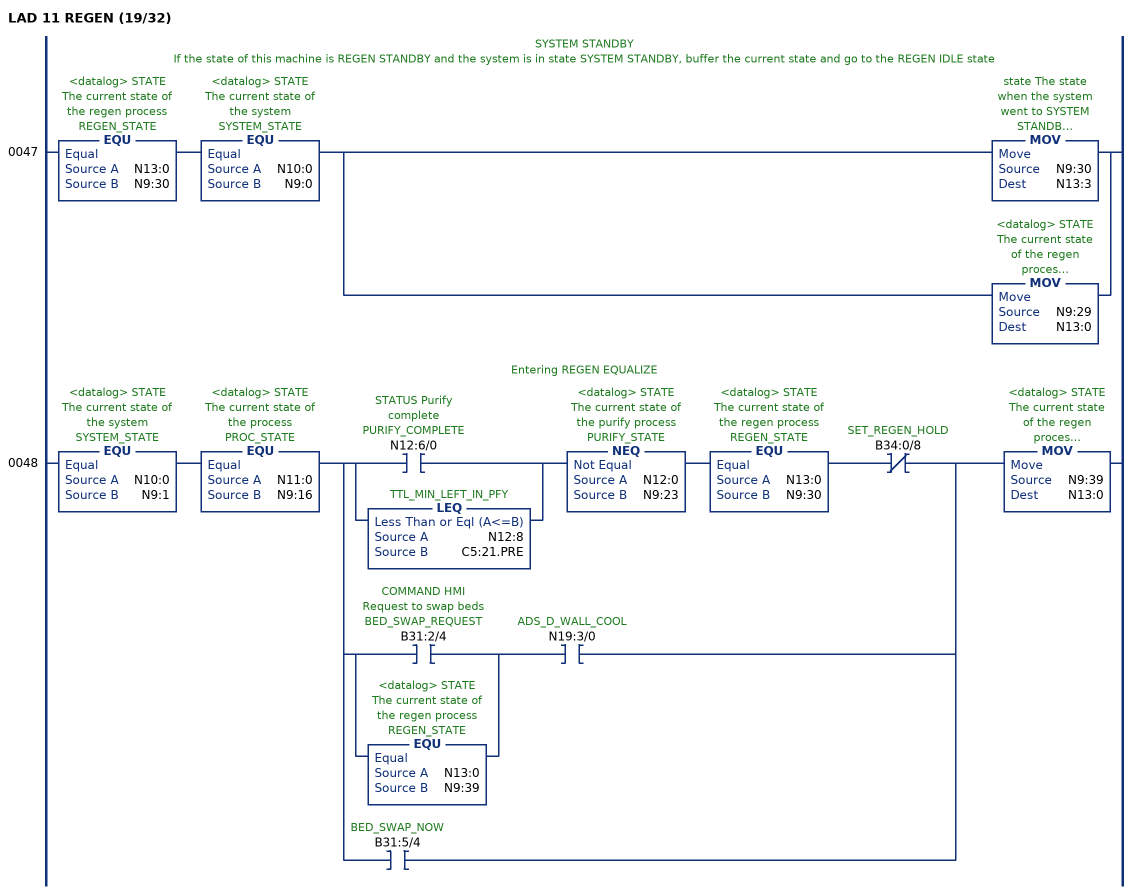
% Rung: 47 %
% SYSTEM STANDBY
% If the state of this machine is REGEN STANDBY and the system is in state SYSTEM STANDBY, buffer the current state and go to the REGEN IDLE state %
SOR EQU N13:0 N9:30 EQU N10:0 N9:0 BST MOV N9:30 N13:3 NXB MOV N9:29 N13:0 BND EOR
%   N13:0  REGEN_STATE  "<datalog> STATE The current state of the regen process" %
%   N9:30  REGEN_STANDBY  "STATE Regen Standby" %
%   N10:0  SYSTEM_STATE  "<datalog> STATE The current state of the system" %
%   N9:0  SYSTEM_STANDBY  "STATE System Standby" %
%   N13:3  REGEN_STANDBY_BUFFER  "state The state when the system went to SYSTEM STANDBY" %
%   N9:29  REGEN_IDLE  "STATE Regen Idle" %
% Rung: 48 %
% Entering REGEN EQUALIZE %
SOR EQU N10:0 N9:1 EQU N11:0 N9:16 BST BST XIC N12:6/0 NXB LEQ N12:8 C5:21.PRE BND NEQ N12:0 N9:23 EQU N13:0 N9:30 XIO B34:0/8 NXB BST XIC B31:2/4 NXB EQU N13:0 N9:39 BND XIC N19:3/0 NXB XIC B31:5/4 BND MOV N9:39 N13:0 EOR
%   N10:0  SYSTEM_STATE  "<datalog> STATE The current state of the system" %
%   N9:1  SYSTEM_PROCESS  "STATE System Process" %
%   N11:0  PROC_STATE  "<datalog> STATE The current state of the process" %
%   N9:16  PROC_REGEN_D  "STATE Process Regen D" %
%   N12:6/0  PURIFY_COMPLETE  "STATUS Purify complete" %
%   N12:8  TTL_MIN_LEFT_IN_PFY %
%   C5:21.PRE  "COUNTER Regen Equalize Time" %
%   N12:0  PURIFY_STATE  "<datalog> STATE The current state of the purify process" %
%   N9:23  PURIFY_MANUAL_HOLD  "STATE Purify Manual Hold" %
%   N13:0  REGEN_STATE  "<datalog> STATE The current state of the regen process" %
%   N9:30  REGEN_STANDBY  "STATE Regen Standby" %
%   B34:0/8  SET_REGEN_HOLD %
%   B31:2/4  BED_SWAP_REQUEST  "COMMAND HMI Request to swap beds" %
%   N9:39  REGEN_EQUALIZE  "STATE Regen Equalize" %
%   N19:3/0  ADS_D_WALL_COOL %
%   B31:5/4  BED_SWAP_NOW %

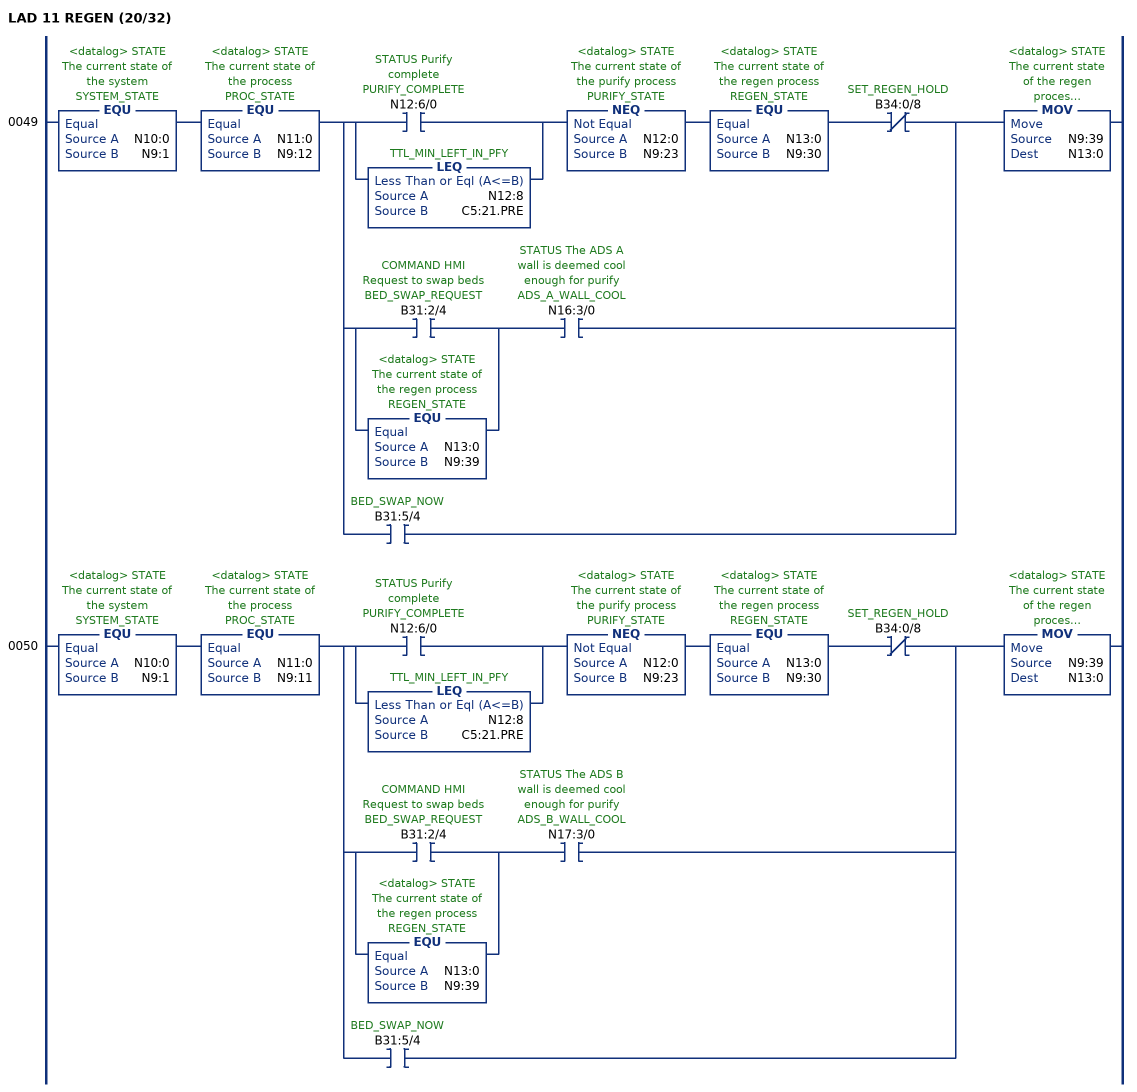
% Rung: 49 %
SOR EQU N10:0 N9:1 EQU N11:0 N9:12 BST BST XIC N12:6/0 NXB LEQ N12:8 C5:21.PRE BND NEQ N12:0 N9:23 EQU N13:0 N9:30 XIO B34:0/8 NXB BST XIC B31:2/4 NXB EQU N13:0 N9:39 BND XIC N16:3/0 NXB XIC B31:5/4 BND MOV N9:39 N13:0 EOR
%   N10:0  SYSTEM_STATE  "<datalog> STATE The current state of the system" %
%   N9:1  SYSTEM_PROCESS  "STATE System Process" %
%   N11:0  PROC_STATE  "<datalog> STATE The current state of the process" %
%   N9:12  PROC_REGEN_A  "STATE Process Regen A" %
%   N12:6/0  PURIFY_COMPLETE  "STATUS Purify complete" %
%   N12:8  TTL_MIN_LEFT_IN_PFY %
%   C5:21.PRE  "COUNTER Regen Equalize Time" %
%   N12:0  PURIFY_STATE  "<datalog> STATE The current state of the purify process" %
%   N9:23  PURIFY_MANUAL_HOLD  "STATE Purify Manual Hold" %
%   N13:0  REGEN_STATE  "<datalog> STATE The current state of the regen process" %
%   N9:30  REGEN_STANDBY  "STATE Regen Standby" %
%   B34:0/8  SET_REGEN_HOLD %
%   B31:2/4  BED_SWAP_REQUEST  "COMMAND HMI Request to swap beds" %
%   N9:39  REGEN_EQUALIZE  "STATE Regen Equalize" %
%   N16:3/0  ADS_A_WALL_COOL  "STATUS The ADS A wall is deemed cool enough for purify" %
%   B31:5/4  BED_SWAP_NOW %
% Rung: 50 %
SOR EQU N10:0 N9:1 EQU N11:0 N9:11 BST BST XIC N12:6/0 NXB LEQ N12:8 C5:21.PRE BND NEQ N12:0 N9:23 EQU N13:0 N9:30 XIO B34:0/8 NXB BST XIC B31:2/4 NXB EQU N13:0 N9:39 BND XIC N17:3/0 NXB XIC B31:5/4 BND MOV N9:39 N13:0 EOR
%   N10:0  SYSTEM_STATE  "<datalog> STATE The current state of the system" %
%   N9:1  SYSTEM_PROCESS  "STATE System Process" %
%   N11:0  PROC_STATE  "<datalog> STATE The current state of the process" %
%   N9:11  PROC_REGEN_B  "STATE Process Regen B" %
%   N12:6/0  PURIFY_COMPLETE  "STATUS Purify complete" %
%   N12:8  TTL_MIN_LEFT_IN_PFY %
%   C5:21.PRE  "COUNTER Regen Equalize Time" %
%   N12:0  PURIFY_STATE  "<datalog> STATE The current state of the purify process" %
%   N9:23  PURIFY_MANUAL_HOLD  "STATE Purify Manual Hold" %
%   N13:0  REGEN_STATE  "<datalog> STATE The current state of the regen process" %
%   N9:30  REGEN_STANDBY  "STATE Regen Standby" %
%   B34:0/8  SET_REGEN_HOLD %
%   B31:2/4  BED_SWAP_REQUEST  "COMMAND HMI Request to swap beds" %
%   N9:39  REGEN_EQUALIZE  "STATE Regen Equalize" %
%   N17:3/0  ADS_B_WALL_COOL  "STATUS The ADS B wall is deemed cool enough for purify" %
%   B31:5/4  BED_SWAP_NOW %

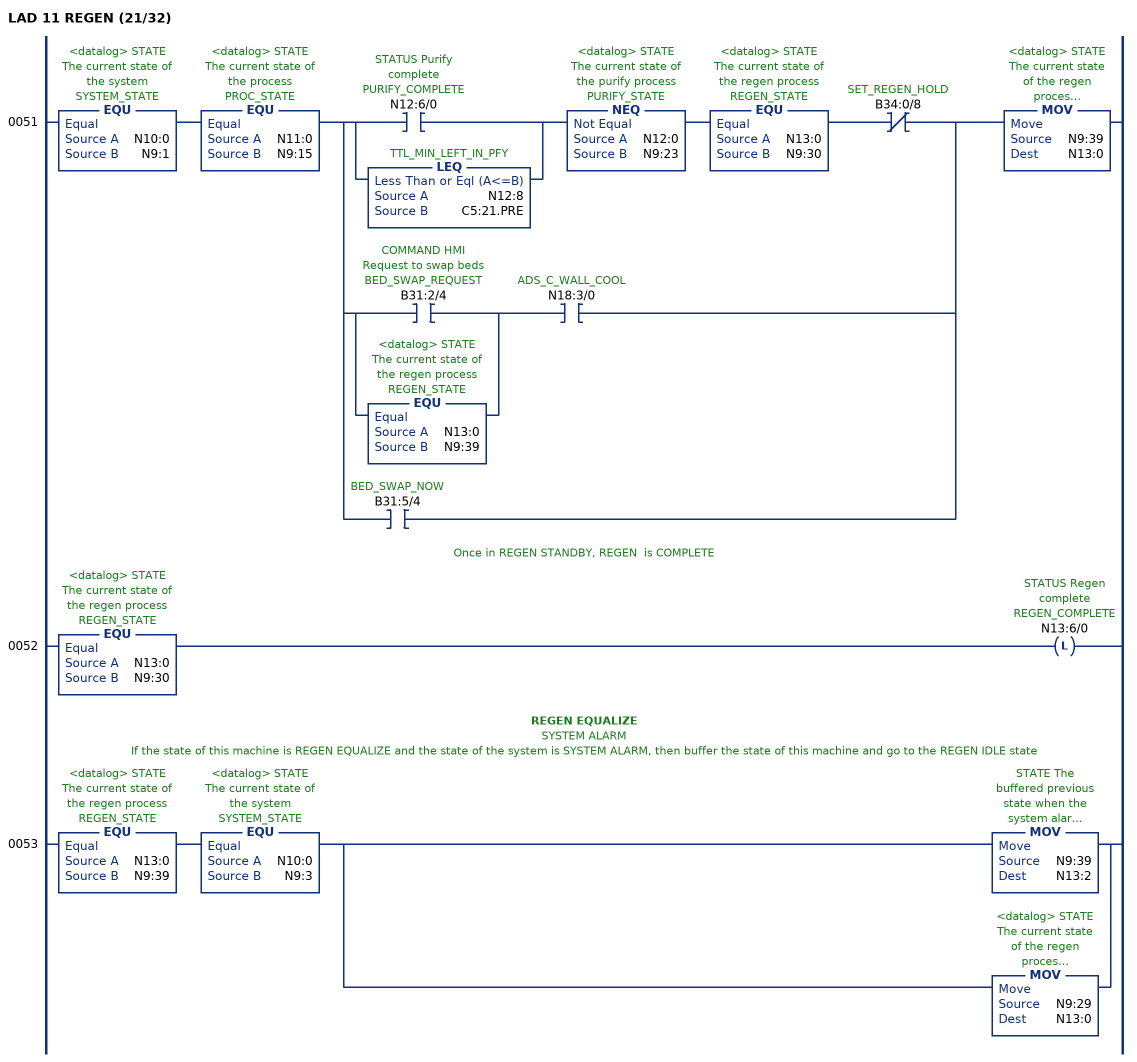
% Rung: 51 %
SOR EQU N10:0 N9:1 EQU N11:0 N9:15 BST BST XIC N12:6/0 NXB LEQ N12:8 C5:21.PRE BND NEQ N12:0 N9:23 EQU N13:0 N9:30 XIO B34:0/8 NXB BST XIC B31:2/4 NXB EQU N13:0 N9:39 BND XIC N18:3/0 NXB XIC B31:5/4 BND MOV N9:39 N13:0 EOR
%   N10:0  SYSTEM_STATE  "<datalog> STATE The current state of the system" %
%   N9:1  SYSTEM_PROCESS  "STATE System Process" %
%   N11:0  PROC_STATE  "<datalog> STATE The current state of the process" %
%   N9:15  PROC_REGEN_C  "STATE Process Regen C" %
%   N12:6/0  PURIFY_COMPLETE  "STATUS Purify complete" %
%   N12:8  TTL_MIN_LEFT_IN_PFY %
%   C5:21.PRE  "COUNTER Regen Equalize Time" %
%   N12:0  PURIFY_STATE  "<datalog> STATE The current state of the purify process" %
%   N9:23  PURIFY_MANUAL_HOLD  "STATE Purify Manual Hold" %
%   N13:0  REGEN_STATE  "<datalog> STATE The current state of the regen process" %
%   N9:30  REGEN_STANDBY  "STATE Regen Standby" %
%   B34:0/8  SET_REGEN_HOLD %
%   B31:2/4  BED_SWAP_REQUEST  "COMMAND HMI Request to swap beds" %
%   N9:39  REGEN_EQUALIZE  "STATE Regen Equalize" %
%   N18:3/0  ADS_C_WALL_COOL %
%   B31:5/4  BED_SWAP_NOW %
% Rung: 52 %
% Once in REGEN STANDBY, REGEN  is COMPLETE %
SOR EQU N13:0 N9:30 OTL N13:6/0 EOR
%   N13:0  REGEN_STATE  "<datalog> STATE The current state of the regen process" %
%   N9:30  REGEN_STANDBY  "STATE Regen Standby" %
%   N13:6/0  REGEN_COMPLETE  "STATUS Regen complete" %
% Rung: 53 %
% TITLE: REGEN EQUALIZE %
% SYSTEM ALARM
% If the state of this machine is REGEN EQUALIZE and the state of the system is SYSTEM ALARM, then buffer the state of this machine and go to the REGEN IDLE state %
SOR EQU N13:0 N9:39 EQU N10:0 N9:3 BST MOV N9:39 N13:2 NXB MOV N9:29 N13:0 BND EOR
%   N13:0  REGEN_STATE  "<datalog> STATE The current state of the regen process" %
%   N9:39  REGEN_EQUALIZE  "STATE Regen Equalize" %
%   N10:0  SYSTEM_STATE  "<datalog> STATE The current state of the system" %
%   N9:3  SYSTEM_ALARM  "STATE System Alarm" %
%   N13:2  REGEN_ALARM_BUFFER  "STATE The buffered previous state when the system alarm occured" %
%   N9:29  REGEN_IDLE  "STATE Regen Idle" %

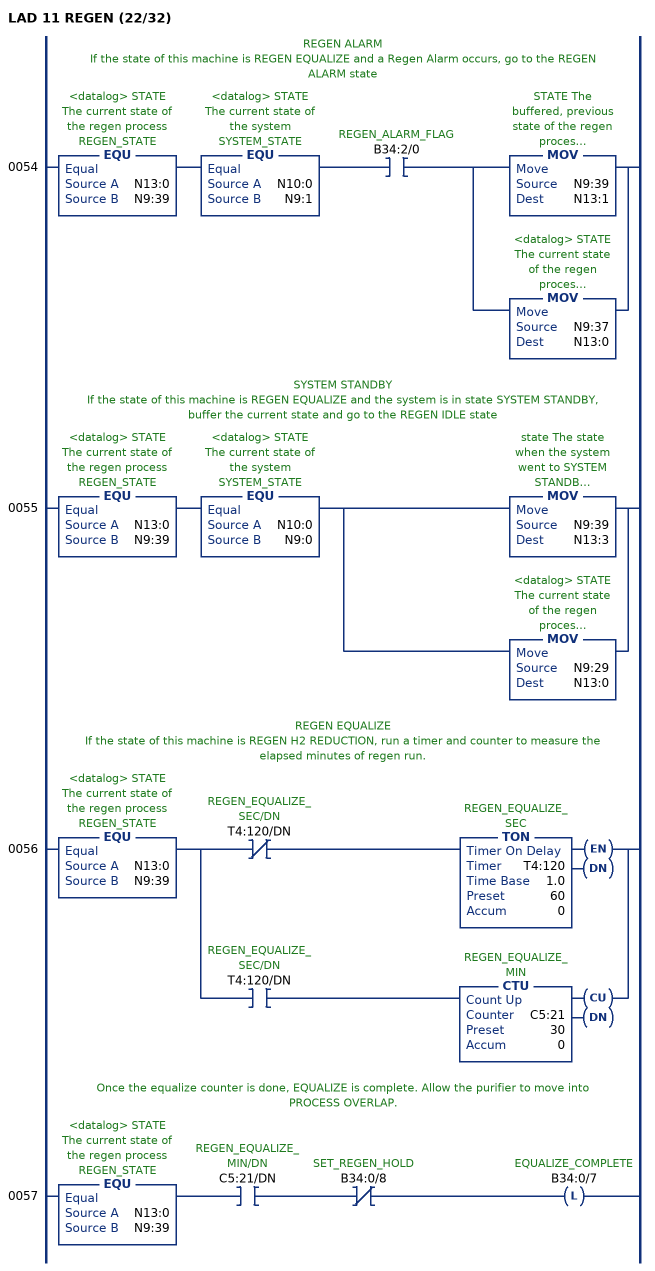
% Rung: 54 %
% REGEN ALARM
% If the state of this machine is REGEN EQUALIZE and a Regen Alarm occurs, go to the REGEN ALARM state %
SOR EQU N13:0 N9:39 EQU N10:0 N9:1 XIC B34:2/0 BST MOV N9:39 N13:1 NXB MOV N9:37 N13:0 BND EOR
%   N13:0  REGEN_STATE  "<datalog> STATE The current state of the regen process" %
%   N9:39  REGEN_EQUALIZE  "STATE Regen Equalize" %
%   N10:0  SYSTEM_STATE  "<datalog> STATE The current state of the system" %
%   N9:1  SYSTEM_PROCESS  "STATE System Process" %
%   B34:2/0  REGEN_ALARM_FLAG %
%   N13:1  REGEN_BUFFER  "STATE The buffered, previous state of the regen process" %
%   N9:37  REGEN_ALARM  "STATE Regen Alarm" %
% Rung: 55 %
% SYSTEM STANDBY
% If the state of this machine is REGEN EQUALIZE and the system is in state SYSTEM STANDBY, buffer the current state and go to the REGEN IDLE state %
SOR EQU N13:0 N9:39 EQU N10:0 N9:0 BST MOV N9:39 N13:3 NXB MOV N9:29 N13:0 BND EOR
%   N13:0  REGEN_STATE  "<datalog> STATE The current state of the regen process" %
%   N9:39  REGEN_EQUALIZE  "STATE Regen Equalize" %
%   N10:0  SYSTEM_STATE  "<datalog> STATE The current state of the system" %
%   N9:0  SYSTEM_STANDBY  "STATE System Standby" %
%   N13:3  REGEN_STANDBY_BUFFER  "state The state when the system went to SYSTEM STANDBY" %
%   N9:29  REGEN_IDLE  "STATE Regen Idle" %
% Rung: 56 %
% REGEN EQUALIZE
% If the state of this machine is REGEN H2 REDUCTION, run a timer and counter to measure the elapsed minutes of regen run. %
SOR EQU N13:0 N9:39 BST XIO T4:120/DN TON T4:120 1.0 60 0 NXB XIC T4:120/DN CTU C5:21 30 0 BND EOR
%   N13:0  REGEN_STATE  "<datalog> STATE The current state of the regen process" %
%   N9:39  REGEN_EQUALIZE  "STATE Regen Equalize" %
%   T4:120  REGEN_EQUALIZE_SEC %
%   C5:21  REGEN_EQUALIZE_MIN %
% Rung: 57 %
% Once the equalize counter is done, EQUALIZE is complete. Allow the purifier to move into PROCESS OVERLAP. %
SOR EQU N13:0 N9:39 XIC C5:21/DN XIO B34:0/8 OTL B34:0/7 EOR
%   N13:0  REGEN_STATE  "<datalog> STATE The current state of the regen process" %
%   N9:39  REGEN_EQUALIZE  "STATE Regen Equalize" %
%   C5:21  REGEN_EQUALIZE_MIN %
%   B34:0/8  SET_REGEN_HOLD %
%   B34:0/7  EQUALIZE_COMPLETE %

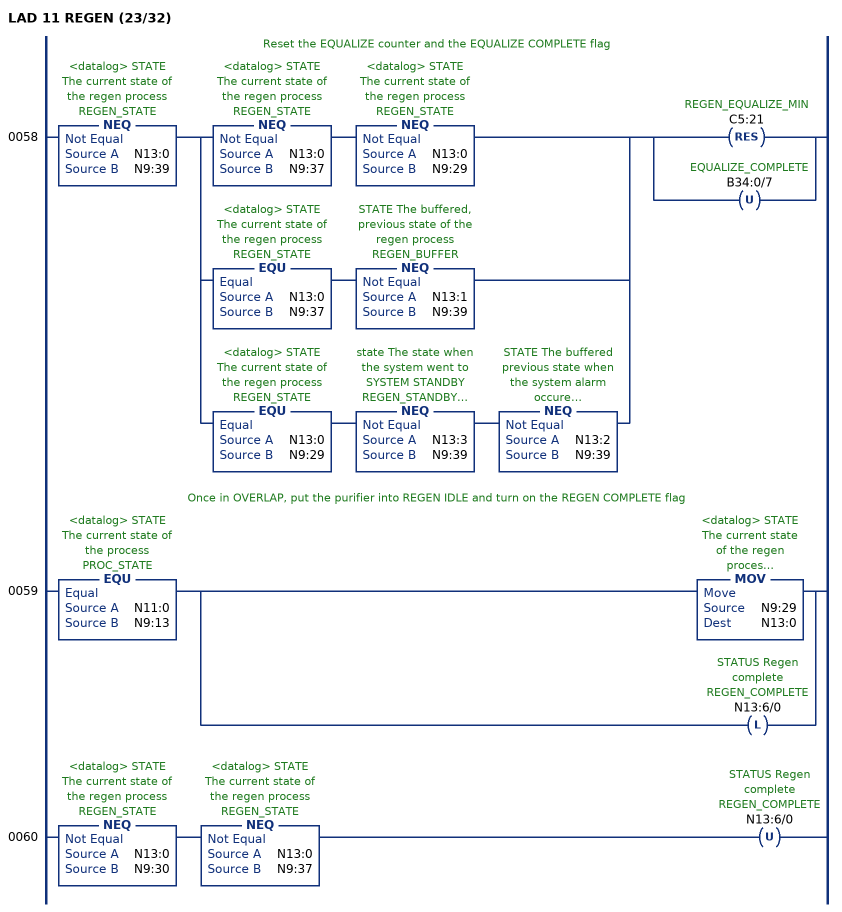
% Rung: 58 %
% Reset the EQUALIZE counter and the EQUALIZE COMPLETE flag %
SOR NEQ N13:0 N9:39 BST NEQ N13:0 N9:37 NEQ N13:0 N9:29 NXB EQU N13:0 N9:37 NEQ N13:1 N9:39 NXB EQU N13:0 N9:29 NEQ N13:3 N9:39 NEQ N13:2 N9:39 BND BST RES C5:21 NXB OTU B34:0/7 BND EOR
%   N13:0  REGEN_STATE  "<datalog> STATE The current state of the regen process" %
%   N9:39  REGEN_EQUALIZE  "STATE Regen Equalize" %
%   N9:37  REGEN_ALARM  "STATE Regen Alarm" %
%   N9:29  REGEN_IDLE  "STATE Regen Idle" %
%   N13:1  REGEN_BUFFER  "STATE The buffered, previous state of the regen process" %
%   N13:3  REGEN_STANDBY_BUFFER  "state The state when the system went to SYSTEM STANDBY" %
%   N13:2  REGEN_ALARM_BUFFER  "STATE The buffered previous state when the system alarm occured" %
%   C5:21  REGEN_EQUALIZE_MIN %
%   B34:0/7  EQUALIZE_COMPLETE %
% Rung: 59 %
% Once in OVERLAP, put the purifier into REGEN IDLE and turn on the REGEN COMPLETE flag %
SOR EQU N11:0 N9:13 BST MOV N9:29 N13:0 NXB OTL N13:6/0 BND EOR
%   N11:0  PROC_STATE  "<datalog> STATE The current state of the process" %
%   N9:13  PROC_OVERLAP  "STATE Process Purify Overlap" %
%   N9:29  REGEN_IDLE  "STATE Regen Idle" %
%   N13:0  REGEN_STATE  "<datalog> STATE The current state of the regen process" %
%   N13:6/0  REGEN_COMPLETE  "STATUS Regen complete" %
% Rung: 60 %
SOR NEQ N13:0 N9:30 NEQ N13:0 N9:37 OTU N13:6/0 EOR
%   N13:0  REGEN_STATE  "<datalog> STATE The current state of the regen process" %
%   N9:30  REGEN_STANDBY  "STATE Regen Standby" %
%   N9:37  REGEN_ALARM  "STATE Regen Alarm" %
%   N13:6/0  REGEN_COMPLETE  "STATUS Regen complete" %

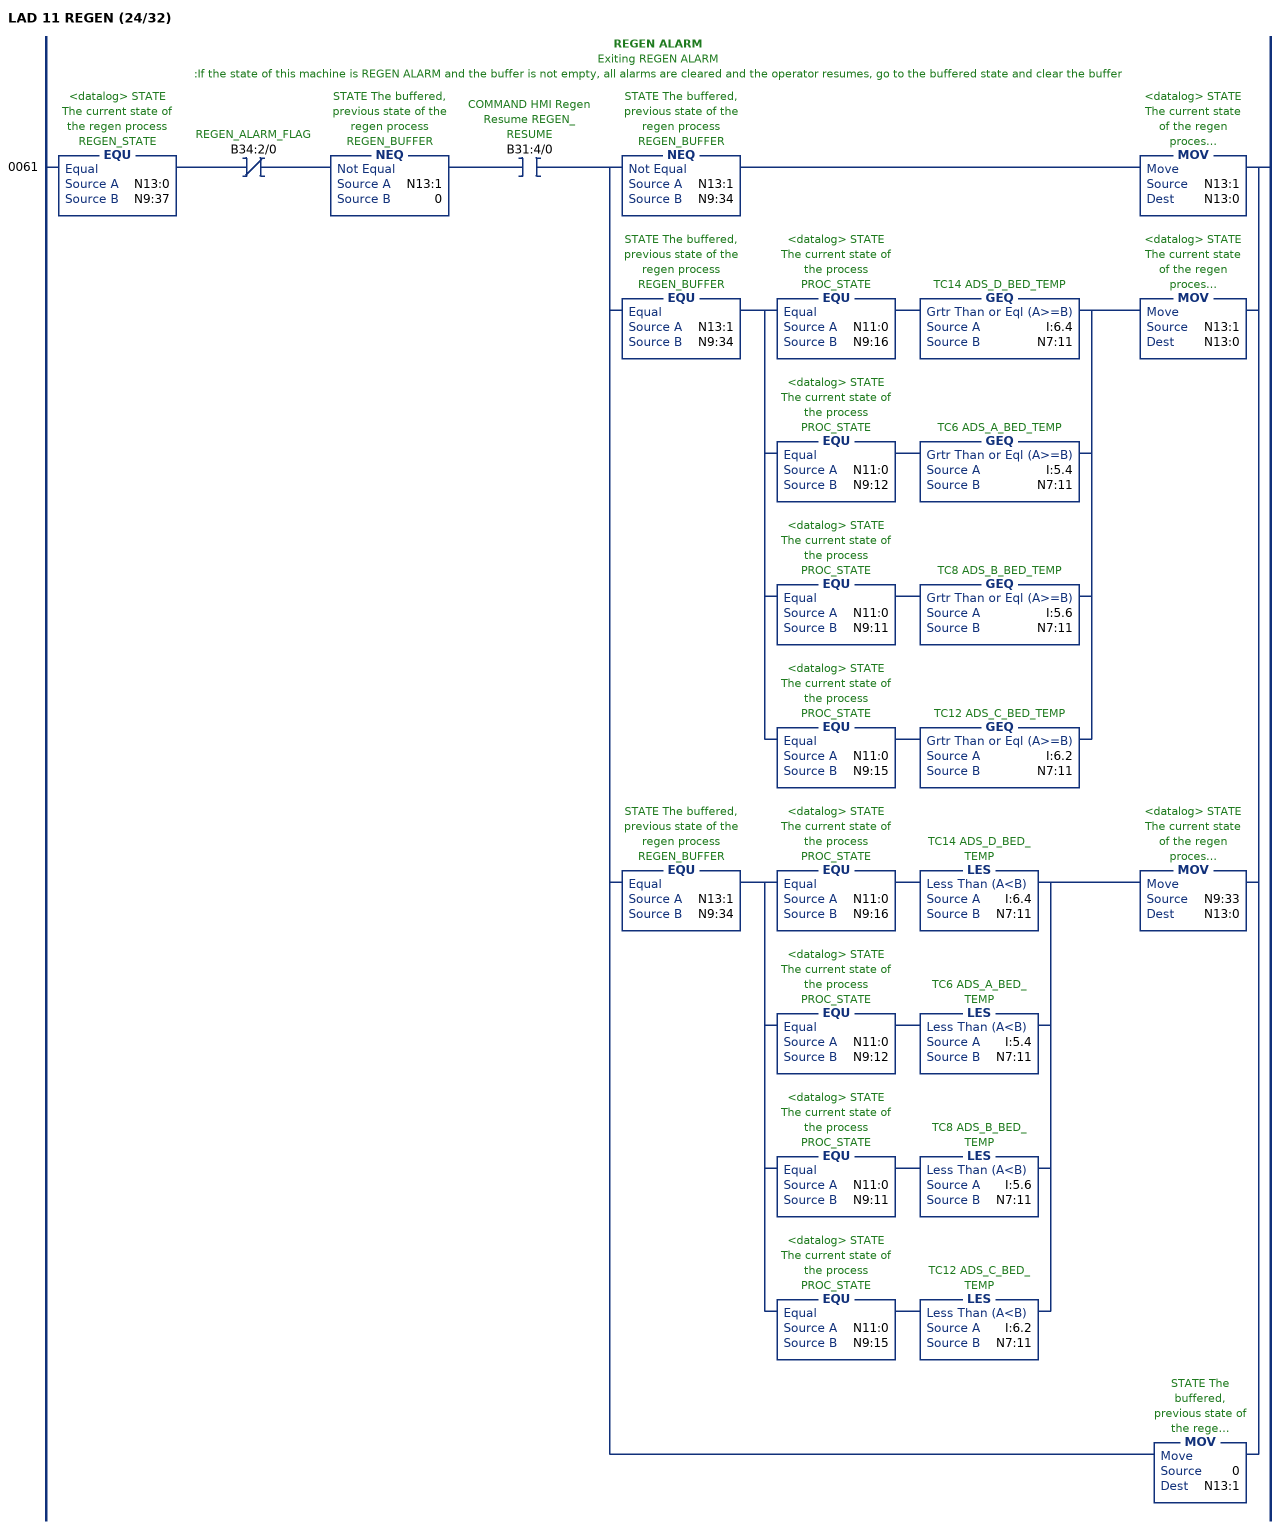
% Rung: 61 %
% TITLE: REGEN ALARM %
% Exiting REGEN ALARM
% :If the state of this machine is REGEN ALARM and the buffer is not empty, all alarms are cleared and the operator resumes, go to the buffered state and clear the buffer %
SOR EQU N13:0 N9:37 XIO B34:2/0 NEQ N13:1 0 XIC B31:4/0 BST NEQ N13:1 N9:34 MOV N13:1 N13:0 NXB EQU N13:1 N9:34 BST EQU N11:0 N9:16 GEQ I:6.4 N7:11 NXB EQU N11:0 N9:12 GEQ I:5.4 N7:11 NXB EQU N11:0 N9:11 GEQ I:5.6 N7:11 NXB EQU N11:0 N9:15 GEQ I:6.2 N7:11 BND MOV N13:1 N13:0 NXB EQU N13:1 N9:34 BST EQU N11:0 N9:16 LES I:6.4 N7:11 NXB EQU N11:0 N9:12 LES I:5.4 N7:11 NXB EQU N11:0 N9:11 LES I:5.6 N7:11 NXB EQU N11:0 N9:15 LES I:6.2 N7:11 BND MOV N9:33 N13:0 NXB MOV 0 N13:1 BND EOR
%   N13:0  REGEN_STATE  "<datalog> STATE The current state of the regen process" %
%   N9:37  REGEN_ALARM  "STATE Regen Alarm" %
%   B34:2/0  REGEN_ALARM_FLAG %
%   N13:1  REGEN_BUFFER  "STATE The buffered, previous state of the regen process" %
%   B31:4/0  REGEN_RESUME  "COMMAND HMI Regen Resume" %
%   N9:34  REGEN_H2_REDUCTION  "STATE Regen Running" %
%   N11:0  PROC_STATE  "<datalog> STATE The current state of the process" %
%   N9:16  PROC_REGEN_D  "STATE Process Regen D" %
%   I:6.4  ADS_D_BED_TEMP  "TC14" %
%   N7:11  ADS_BED_TEMP_HIGH  "CONFIG The temp at which the regen process may continue" %
%   N9:12  PROC_REGEN_A  "STATE Process Regen A" %
%   I:5.4  ADS_A_BED_TEMP  "TC6" %
%   N9:11  PROC_REGEN_B  "STATE Process Regen B" %
%   I:5.6  ADS_B_BED_TEMP  "TC8" %
%   N9:15  PROC_REGEN_C  "STATE Process Regen C" %
%   I:6.2  ADS_C_BED_TEMP  "TC12" %
%   N9:33  REGEN_HEAT_BED  "STATE Regen Heat wall" %

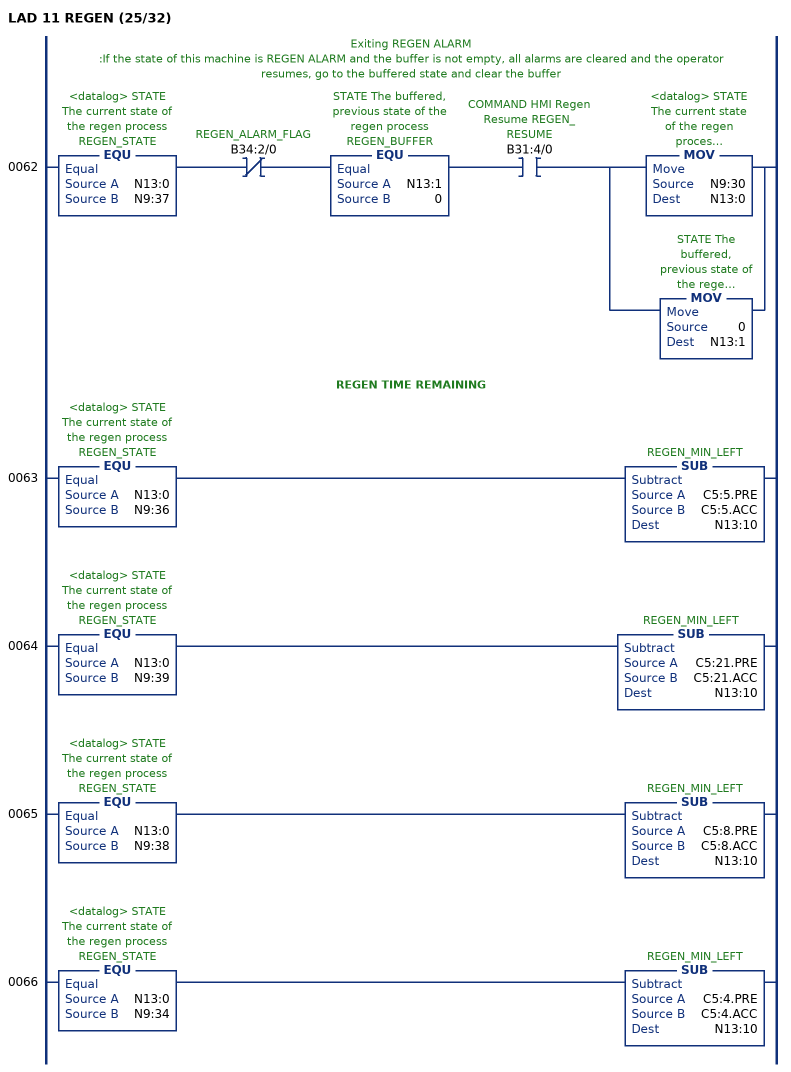
% Rung: 62 %
% Exiting REGEN ALARM
% :If the state of this machine is REGEN ALARM and the buffer is not empty, all alarms are cleared and the operator resumes, go to the buffered state and clear the buffer %
SOR EQU N13:0 N9:37 XIO B34:2/0 EQU N13:1 0 XIC B31:4/0 BST MOV N9:30 N13:0 NXB MOV 0 N13:1 BND EOR
%   N13:0  REGEN_STATE  "<datalog> STATE The current state of the regen process" %
%   N9:37  REGEN_ALARM  "STATE Regen Alarm" %
%   B34:2/0  REGEN_ALARM_FLAG %
%   N13:1  REGEN_BUFFER  "STATE The buffered, previous state of the regen process" %
%   B31:4/0  REGEN_RESUME  "COMMAND HMI Regen Resume" %
%   N9:30  REGEN_STANDBY  "STATE Regen Standby" %
% Rung: 63 %
% TITLE: REGEN TIME REMAINING %
SOR EQU N13:0 N9:36 SUB C5:5.PRE C5:5.ACC N13:10 EOR
%   N13:0  REGEN_STATE  "<datalog> STATE The current state of the regen process" %
%   N9:36  REGEN_COOL  "STATE Regen Cool" %
%   C5:5  REGEN_COOL_MINUTE  "COUNTER Regen the number of minutes for which the bed has cooled" %
%   N13:10  REGEN_MIN_LEFT %
% Rung: 64 %
SOR EQU N13:0 N9:39 SUB C5:21.PRE C5:21.ACC N13:10 EOR
%   N13:0  REGEN_STATE  "<datalog> STATE The current state of the regen process" %
%   N9:39  REGEN_EQUALIZE  "STATE Regen Equalize" %
%   C5:21.PRE  "COUNTER Regen Equalize Time" %
%   C5:21  REGEN_EQUALIZE_MIN %
%   N13:10  REGEN_MIN_LEFT %
% Rung: 65 %
SOR EQU N13:0 N9:38 SUB C5:8.PRE C5:8.ACC N13:10 EOR
%   N13:0  REGEN_STATE  "<datalog> STATE The current state of the regen process" %
%   N9:38  REGEN_PURGE  "STATE Regen Hot Purge" %
%   C5:8  REGEN_PURGE_MINUTES  "COUNTER Regen THe number of minutes the purge step runs" %
%   N13:10  REGEN_MIN_LEFT %
% Rung: 66 %
SOR EQU N13:0 N9:34 SUB C5:4.PRE C5:4.ACC N13:10 EOR
%   N13:0  REGEN_STATE  "<datalog> STATE The current state of the regen process" %
%   N9:34  REGEN_H2_REDUCTION  "STATE Regen Running" %
%   C5:4  REGEN_REDUC_MINUTE  "COUNTER Regen The number of minutes which the regen reduc runs" %
%   N13:10  REGEN_MIN_LEFT %

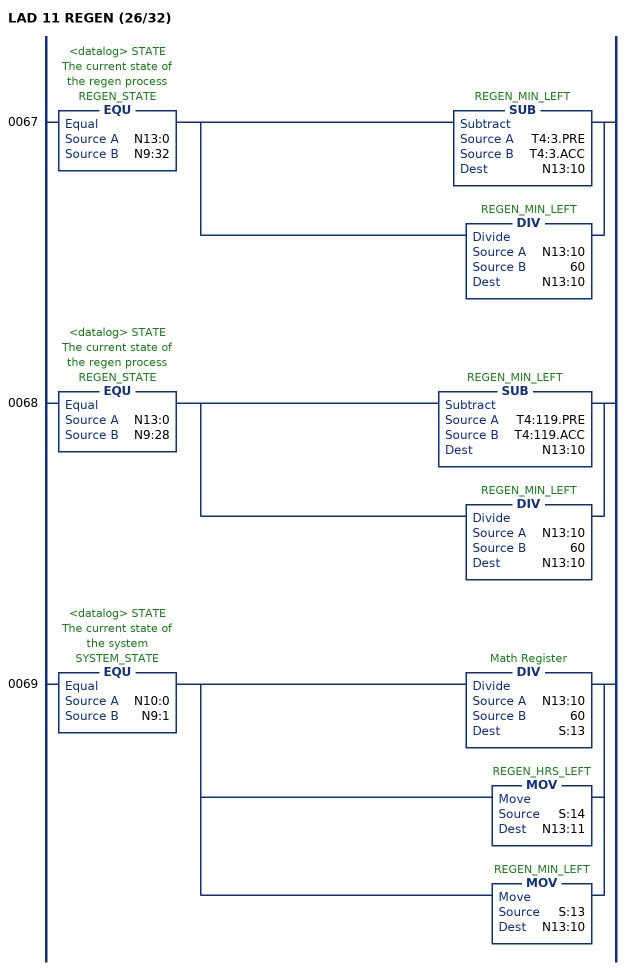
% Rung: 67 %
SOR EQU N13:0 N9:32 BST SUB T4:3.PRE T4:3.ACC N13:10 NXB DIV N13:10 60 N13:10 BND EOR
%   N13:0  REGEN_STATE  "<datalog> STATE The current state of the regen process" %
%   N9:32  REGEN_VENT  "STATE Regen Vent" %
%   T4:3  REGEN_VENT_TIMER  "TIMER Regen Vent (seconds)" %
%   N13:10  REGEN_MIN_LEFT %
% Rung: 68 %
SOR EQU N13:0 N9:28 BST SUB T4:119.PRE T4:119.ACC N13:10 NXB DIV N13:10 60 N13:10 BND EOR
%   N13:0  REGEN_STATE  "<datalog> STATE The current state of the regen process" %
%   N9:28  REGEN_VENT_2 %
%   T4:119  REGEN_VENT_2_TMR %
%   N13:10  REGEN_MIN_LEFT %
% Rung: 69 %
SOR EQU N10:0 N9:1 BST DIV N13:10 60 S:13 NXB MOV S:14 N13:11 NXB MOV S:13 N13:10 BND EOR
%   N10:0  SYSTEM_STATE  "<datalog> STATE The current state of the system" %
%   N9:1  SYSTEM_PROCESS  "STATE System Process" %
%   N13:10  REGEN_MIN_LEFT %
%   S:13  "Math Register" %
%   S:14  "Math Register" %
%   N13:11  REGEN_HRS_LEFT %

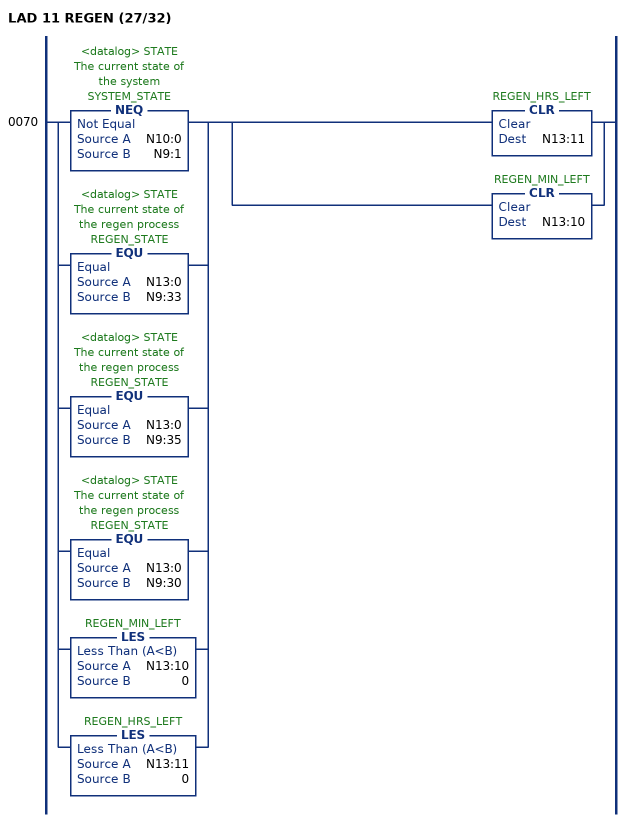
% Rung: 70 %
SOR BST NEQ N10:0 N9:1 NXB EQU N13:0 N9:33 NXB EQU N13:0 N9:35 NXB EQU N13:0 N9:30 NXB LES N13:10 0 NXB LES N13:11 0 BND BST CLR N13:11 NXB CLR N13:10 BND EOR
%   N10:0  SYSTEM_STATE  "<datalog> STATE The current state of the system" %
%   N9:1  SYSTEM_PROCESS  "STATE System Process" %
%   N13:0  REGEN_STATE  "<datalog> STATE The current state of the regen process" %
%   N9:33  REGEN_HEAT_BED  "STATE Regen Heat wall" %
%   N9:35  REGEN_COOL_WALL  "STATE Regen Cool wall" %
%   N9:30  REGEN_STANDBY  "STATE Regen Standby" %
%   N13:10  REGEN_MIN_LEFT %
%   N13:11  REGEN_HRS_LEFT %

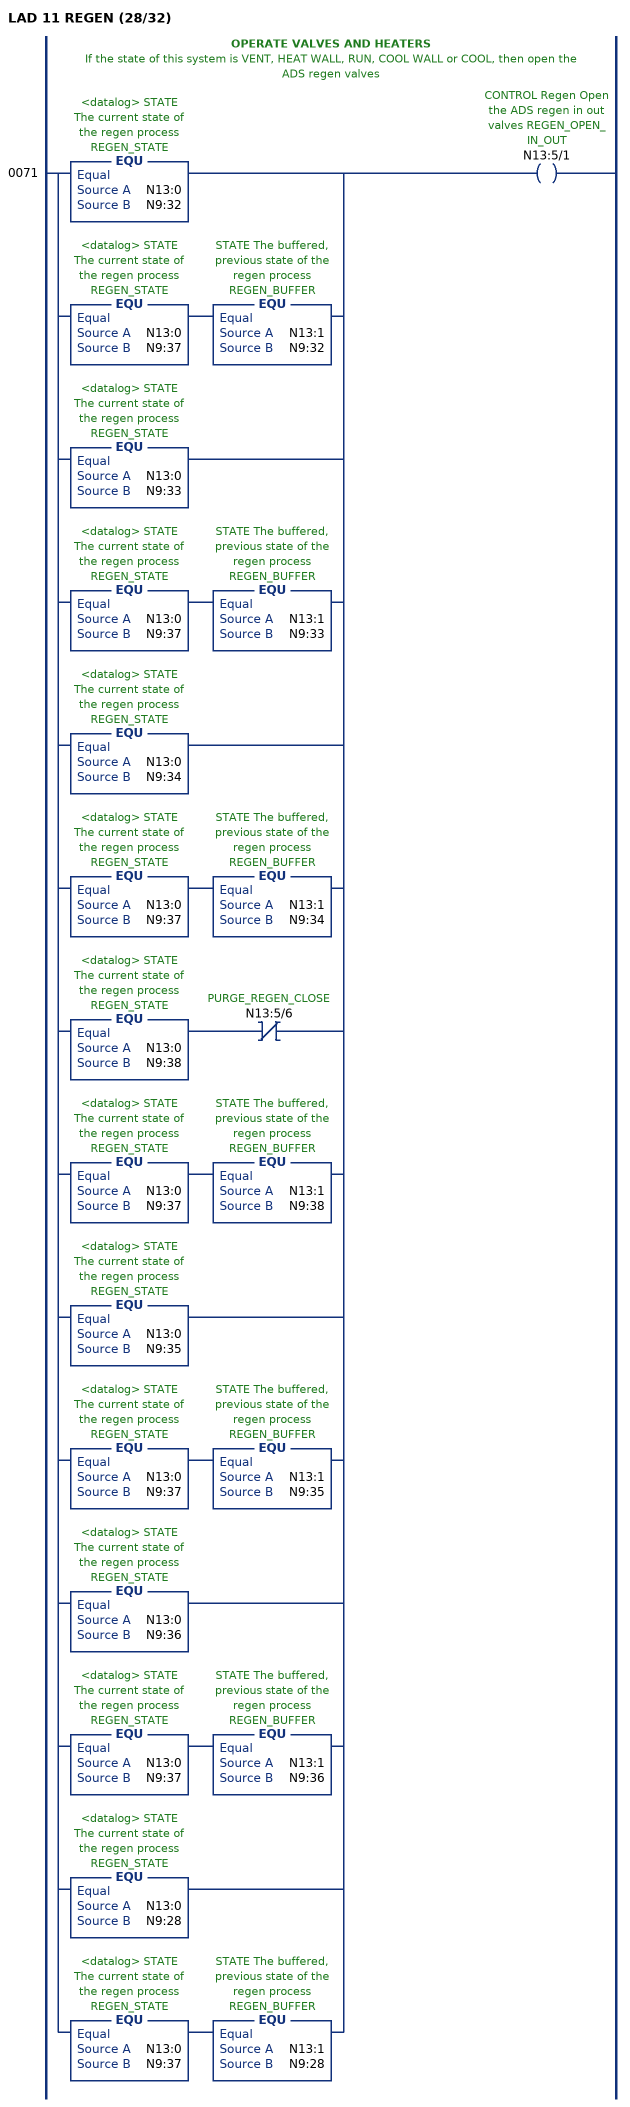
% Rung: 71 %
% TITLE: OPERATE VALVES AND HEATERS %
% If the state of this system is VENT, HEAT WALL, RUN, COOL WALL or COOL, then open the ADS regen valves %
SOR BST EQU N13:0 N9:32 NXB EQU N13:0 N9:37 EQU N13:1 N9:32 NXB EQU N13:0 N9:33 NXB EQU N13:0 N9:37 EQU N13:1 N9:33 NXB EQU N13:0 N9:34 NXB EQU N13:0 N9:37 EQU N13:1 N9:34 NXB EQU N13:0 N9:38 XIO N13:5/6 NXB EQU N13:0 N9:37 EQU N13:1 N9:38 NXB EQU N13:0 N9:35 NXB EQU N13:0 N9:37 EQU N13:1 N9:35 NXB EQU N13:0 N9:36 NXB EQU N13:0 N9:37 EQU N13:1 N9:36 NXB EQU N13:0 N9:28 NXB EQU N13:0 N9:37 EQU N13:1 N9:28 BND OTE N13:5/1 EOR
%   N13:0  REGEN_STATE  "<datalog> STATE The current state of the regen process" %
%   N9:32  REGEN_VENT  "STATE Regen Vent" %
%   N9:37  REGEN_ALARM  "STATE Regen Alarm" %
%   N13:1  REGEN_BUFFER  "STATE The buffered, previous state of the regen process" %
%   N9:33  REGEN_HEAT_BED  "STATE Regen Heat wall" %
%   N9:34  REGEN_H2_REDUCTION  "STATE Regen Running" %
%   N9:38  REGEN_PURGE  "STATE Regen Hot Purge" %
%   N13:5/6  PURGE_REGEN_CLOSE %
%   N9:35  REGEN_COOL_WALL  "STATE Regen Cool wall" %
%   N9:36  REGEN_COOL  "STATE Regen Cool" %
%   N9:28  REGEN_VENT_2 %
%   N13:5/1  REGEN_OPEN_IN_OUT  "CONTROL Regen Open the ADS regen in out valves" %

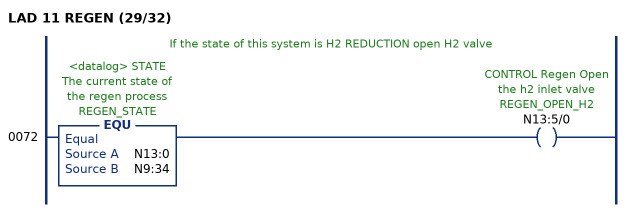
% Rung: 72 %
% If the state of this system is H2 REDUCTION open H2 valve %
SOR EQU N13:0 N9:34 OTE N13:5/0 EOR
%   N13:0  REGEN_STATE  "<datalog> STATE The current state of the regen process" %
%   N9:34  REGEN_H2_REDUCTION  "STATE Regen Running" %
%   N13:5/0  REGEN_OPEN_H2  "CONTROL Regen Open the h2 inlet valve" %

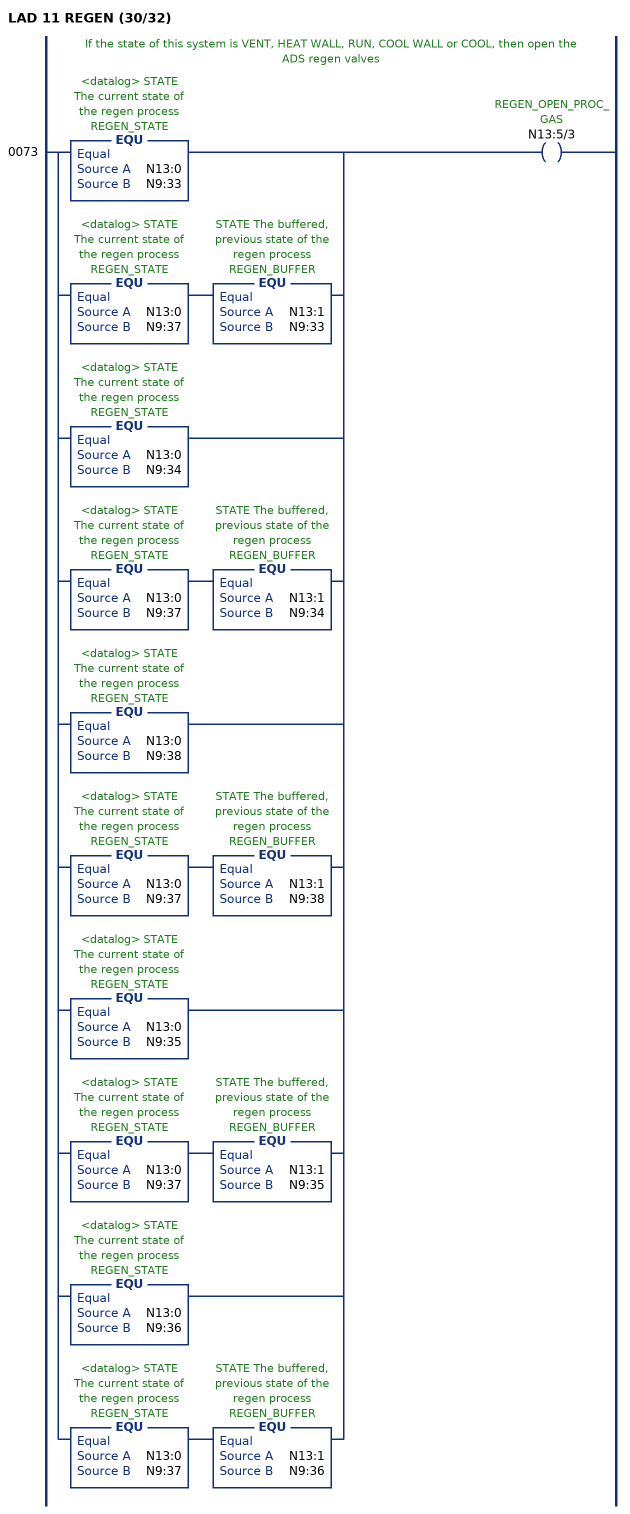
% Rung: 73 %
% If the state of this system is VENT, HEAT WALL, RUN, COOL WALL or COOL, then open the ADS regen valves %
SOR BST EQU N13:0 N9:33 NXB EQU N13:0 N9:37 EQU N13:1 N9:33 NXB EQU N13:0 N9:34 NXB EQU N13:0 N9:37 EQU N13:1 N9:34 NXB EQU N13:0 N9:38 NXB EQU N13:0 N9:37 EQU N13:1 N9:38 NXB EQU N13:0 N9:35 NXB EQU N13:0 N9:37 EQU N13:1 N9:35 NXB EQU N13:0 N9:36 NXB EQU N13:0 N9:37 EQU N13:1 N9:36 BND OTE N13:5/3 EOR
%   N13:0  REGEN_STATE  "<datalog> STATE The current state of the regen process" %
%   N9:33  REGEN_HEAT_BED  "STATE Regen Heat wall" %
%   N9:37  REGEN_ALARM  "STATE Regen Alarm" %
%   N13:1  REGEN_BUFFER  "STATE The buffered, previous state of the regen process" %
%   N9:34  REGEN_H2_REDUCTION  "STATE Regen Running" %
%   N9:38  REGEN_PURGE  "STATE Regen Hot Purge" %
%   N9:35  REGEN_COOL_WALL  "STATE Regen Cool wall" %
%   N9:36  REGEN_COOL  "STATE Regen Cool" %
%   N13:5/3  REGEN_OPEN_PROC_GAS %

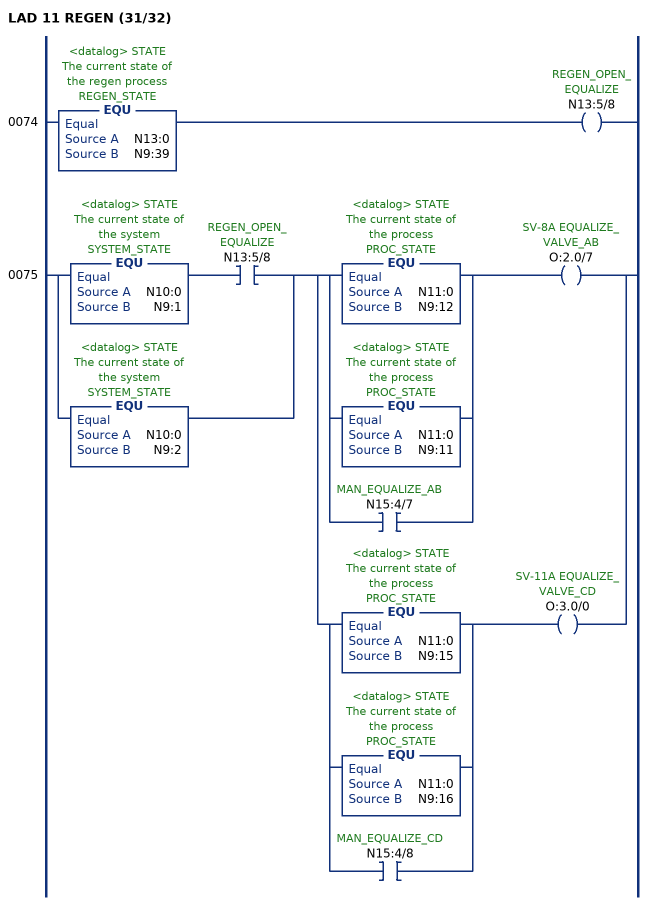
% Rung: 74 %
SOR EQU N13:0 N9:39 OTE N13:5/8 EOR
%   N13:0  REGEN_STATE  "<datalog> STATE The current state of the regen process" %
%   N9:39  REGEN_EQUALIZE  "STATE Regen Equalize" %
%   N13:5/8  REGEN_OPEN_EQUALIZE %
% Rung: 75 %
SOR BST EQU N10:0 N9:1 XIC N13:5/8 NXB EQU N10:0 N9:2 BND BST BST EQU N11:0 N9:12 NXB EQU N11:0 N9:11 NXB XIC N15:4/7 BND OTE O:2.0/7 NXB BST EQU N11:0 N9:15 NXB EQU N11:0 N9:16 NXB XIC N15:4/8 BND OTE O:3.0/0 BND EOR
%   N10:0  SYSTEM_STATE  "<datalog> STATE The current state of the system" %
%   N9:1  SYSTEM_PROCESS  "STATE System Process" %
%   N13:5/8  REGEN_OPEN_EQUALIZE %
%   N9:2  SYSTEM_MANUAL  "STATE System Manual" %
%   N11:0  PROC_STATE  "<datalog> STATE The current state of the process" %
%   N9:12  PROC_REGEN_A  "STATE Process Regen A" %
%   N9:11  PROC_REGEN_B  "STATE Process Regen B" %
%   N15:4/7  MAN_EQUALIZE_AB %
%   O:2.0/7  EQUALIZE_VALVE_AB  "SV-8A" %
%   N9:15  PROC_REGEN_C  "STATE Process Regen C" %
%   N9:16  PROC_REGEN_D  "STATE Process Regen D" %
%   N15:4/8  MAN_EQUALIZE_CD %
%   O:3.0/0  EQUALIZE_VALVE_CD  "SV-11A" %

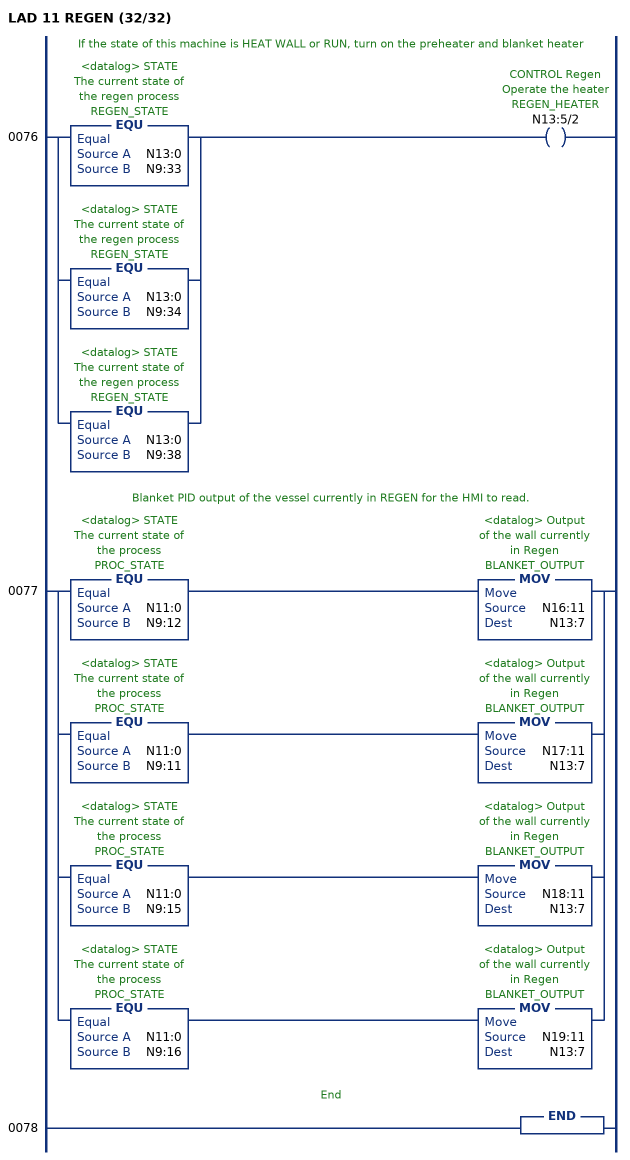
% Rung: 76 %
% If the state of this machine is HEAT WALL or RUN, turn on the preheater and blanket heater %
SOR BST EQU N13:0 N9:33 NXB EQU N13:0 N9:34 NXB EQU N13:0 N9:38 BND OTE N13:5/2 EOR
%   N13:0  REGEN_STATE  "<datalog> STATE The current state of the regen process" %
%   N9:33  REGEN_HEAT_BED  "STATE Regen Heat wall" %
%   N9:34  REGEN_H2_REDUCTION  "STATE Regen Running" %
%   N9:38  REGEN_PURGE  "STATE Regen Hot Purge" %
%   N13:5/2  REGEN_HEATER  "CONTROL Regen Operate the heater" %
% Rung: 77 %
% Blanket PID output of the vessel currently in REGEN for the HMI to read. %
SOR BST EQU N11:0 N9:12 MOV N16:11 N13:7 NXB EQU N11:0 N9:11 MOV N17:11 N13:7 NXB EQU N11:0 N9:15 MOV N18:11 N13:7 NXB EQU N11:0 N9:16 MOV N19:11 N13:7 BND EOR
%   N11:0  PROC_STATE  "<datalog> STATE The current state of the process" %
%   N9:12  PROC_REGEN_A  "STATE Process Regen A" %
%   N16:11  ADS_A_BLNKT_OUTPUT  "<datalog> CONTROL ADS A Blanket output (percent)" %
%   N13:7  BLANKET_OUTPUT  "<datalog> Output of the wall currently in Regen" %
%   N9:11  PROC_REGEN_B  "STATE Process Regen B" %
%   N17:11  ADS_B_BLNKT_OUTPUT  "<datalog> CONTROL ADS A Blanket output" %
%   N9:15  PROC_REGEN_C  "STATE Process Regen C" %
%   N18:11  ADS_C_BLNKT_OUTPUT  "<datalog>" %
%   N9:16  PROC_REGEN_D  "STATE Process Regen D" %
%   N19:11  ADS_D_BLNKT_OUTPUT  "<datalog>" %
% Rung: 78 %
% End %
SOR END EOR

LADDER 12 "REGEN_FLT"    % regen alarms and warnings %
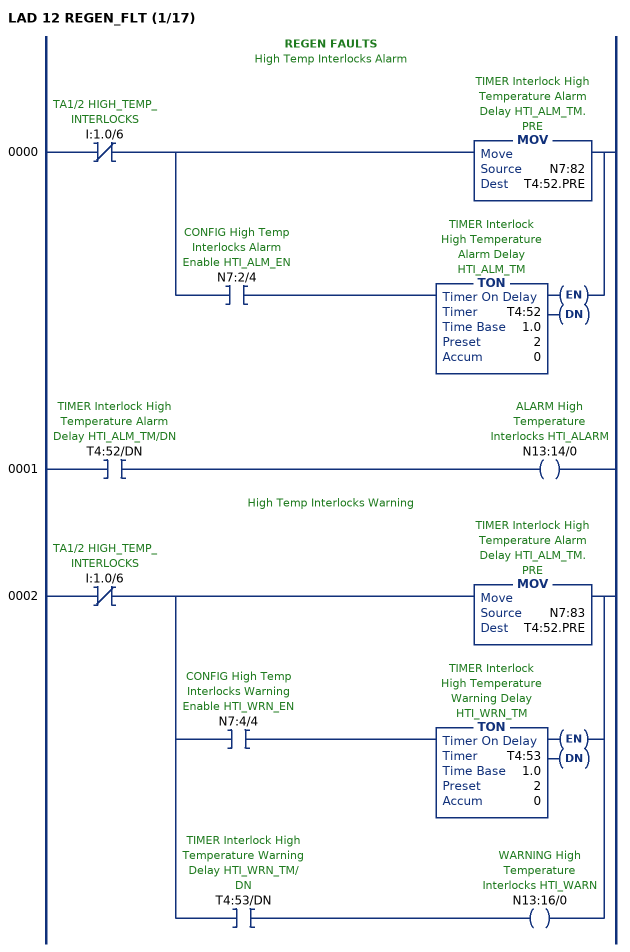
% Rung: 0 %
% TITLE: REGEN FAULTS %
% High Temp Interlocks Alarm %
SOR XIO I:1.0/6 BST MOV N7:82 T4:52.PRE NXB XIC N7:2/4 TON T4:52 1.0 2 0 BND EOR
%   I:1.0/6  HIGH_TEMP_INTERLOCKS  "TA1/2" %
%   N7:82  HTI_ALM_DY  "CONFIG Interlocks High Temp Alarm Delay" %
%   T4:52  HTI_ALM_TM  "TIMER Interlock High Temperature Alarm Delay" %
%   N7:2/4  HTI_ALM_EN  "CONFIG High Temp Interlocks Alarm Enable" %
% Rung: 1 %
SOR XIC T4:52/DN OTE N13:14/0 EOR
%   T4:52  HTI_ALM_TM  "TIMER Interlock High Temperature Alarm Delay" %
%   N13:14/0  HTI_ALARM  "ALARM High Temperature Interlocks" %
% Rung: 2 %
% High Temp Interlocks Warning %
SOR XIO I:1.0/6 BST MOV N7:83 T4:52.PRE NXB XIC N7:4/4 TON T4:53 1.0 2 0 NXB XIC T4:53/DN OTE N13:16/0 BND EOR
%   I:1.0/6  HIGH_TEMP_INTERLOCKS  "TA1/2" %
%   N7:83  HTI_WRN_DY  "CONFIG Interlocks High Temp Warning Delay" %
%   T4:52  HTI_ALM_TM  "TIMER Interlock High Temperature Alarm Delay" %
%   N7:4/4  HTI_WRN_EN  "CONFIG High Temp Interlocks Warning Enable" %
%   T4:53  HTI_WRN_TM  "TIMER Interlock High Temperature Warning Delay" %
%   N13:16/0  HTI_WARN  "WARNING High Temperature Interlocks" %

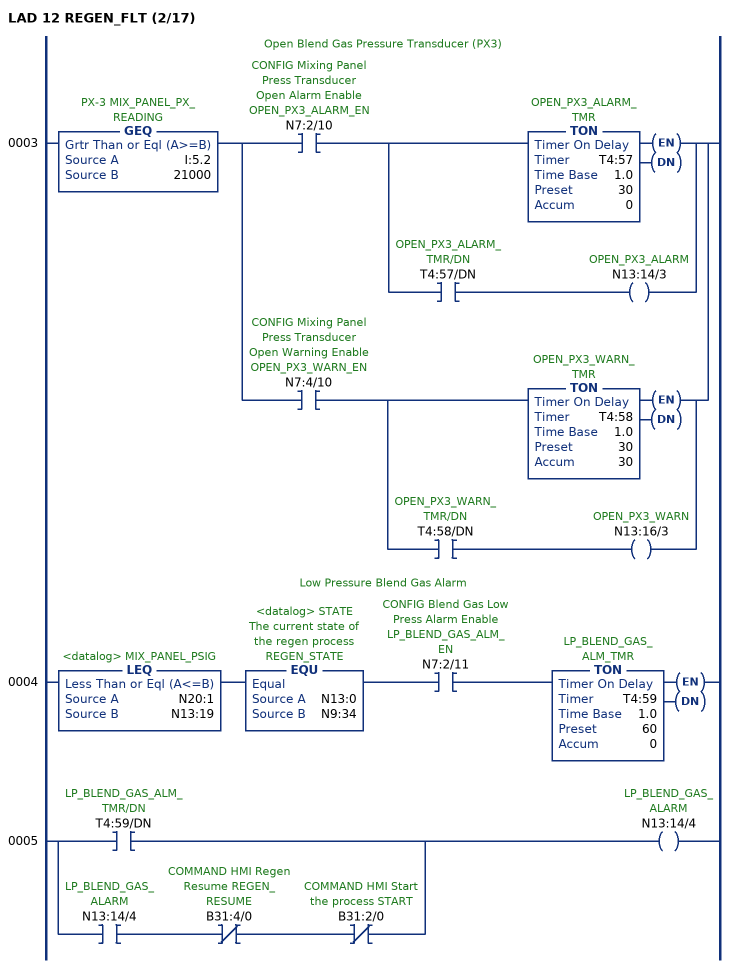
% Rung: 3 %
% Open Blend Gas Pressure Transducer (PX3) %
SOR GEQ I:5.2 21000 BST XIC N7:2/10 BST TON T4:57 1.0 30 0 NXB XIC T4:57/DN OTE N13:14/3 BND NXB XIC N7:4/10 BST TON T4:58 1.0 30 30 NXB XIC T4:58/DN OTE N13:16/3 BND BND EOR
%   I:5.2  MIX_PANEL_PX_READING  "PX-3" %
%   N7:2/10  OPEN_PX3_ALARM_EN  "CONFIG Mixing Panel Press Transducer Open Alarm Enable" %
%   T4:57  OPEN_PX3_ALARM_TMR %
%   N13:14/3  OPEN_PX3_ALARM %
%   N7:4/10  OPEN_PX3_WARN_EN  "CONFIG Mixing Panel Press Transducer Open Warning Enable" %
%   T4:58  OPEN_PX3_WARN_TMR %
%   N13:16/3  OPEN_PX3_WARN %
% Rung: 4 %
% Low Pressure Blend Gas Alarm %
SOR LEQ N20:1 N13:19 EQU N13:0 N9:34 XIC N7:2/11 TON T4:59 1.0 60 0 EOR
%   N20:1  MIX_PANEL_PSIG  "<datalog>" %
%   N13:19  LP_BLEND_GAS_ALM_SP  "CONFIG Blend Gas Low Press Alarm Setpoint" %
%   N13:0  REGEN_STATE  "<datalog> STATE The current state of the regen process" %
%   N9:34  REGEN_H2_REDUCTION  "STATE Regen Running" %
%   N7:2/11  LP_BLEND_GAS_ALM_EN  "CONFIG Blend Gas Low Press Alarm Enable" %
%   T4:59  LP_BLEND_GAS_ALM_TMR %
% Rung: 5 %
SOR BST XIC T4:59/DN NXB XIC N13:14/4 XIO B31:4/0 XIO B31:2/0 BND OTE N13:14/4 EOR
%   T4:59  LP_BLEND_GAS_ALM_TMR %
%   N13:14/4  LP_BLEND_GAS_ALARM %
%   B31:4/0  REGEN_RESUME  "COMMAND HMI Regen Resume" %
%   B31:2/0  START  "COMMAND HMI Start the process" %

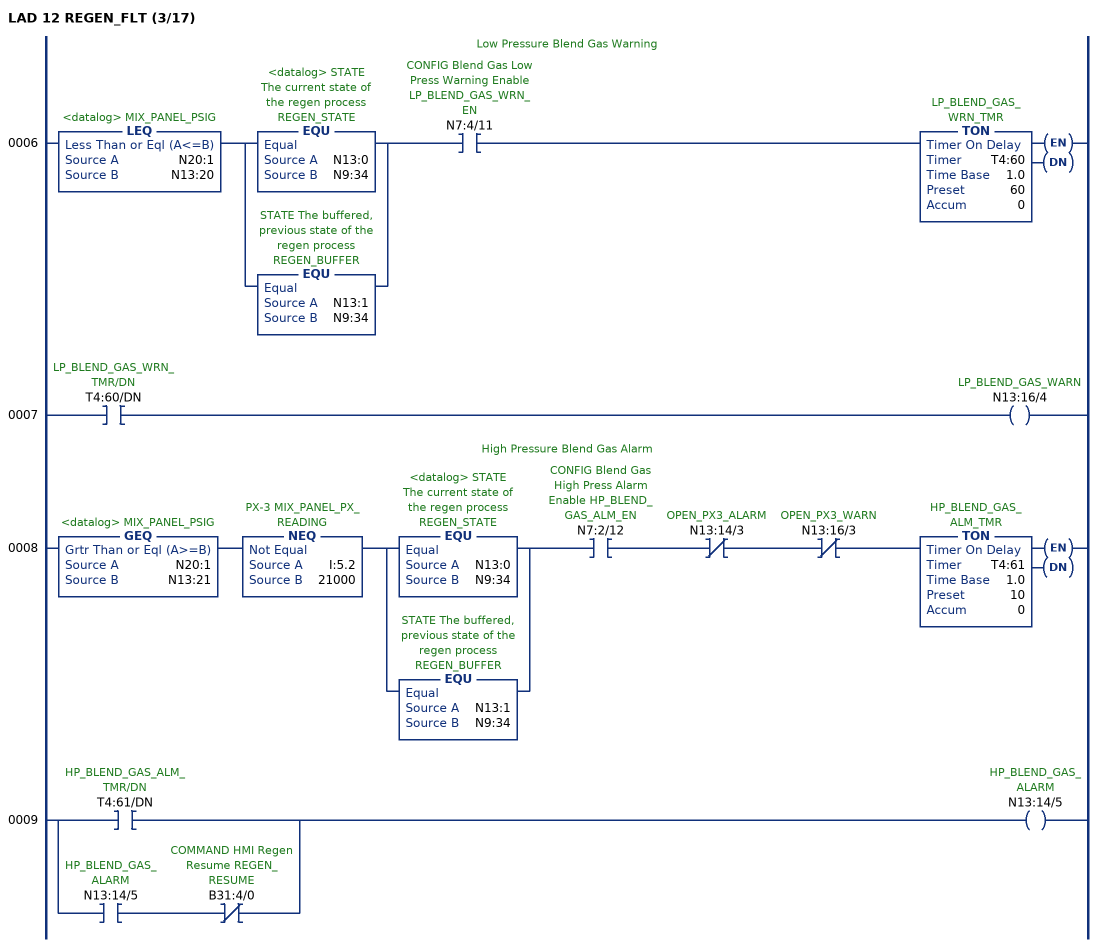
% Rung: 6 %
% Low Pressure Blend Gas Warning %
SOR LEQ N20:1 N13:20 BST EQU N13:0 N9:34 NXB EQU N13:1 N9:34 BND XIC N7:4/11 TON T4:60 1.0 60 0 EOR
%   N20:1  MIX_PANEL_PSIG  "<datalog>" %
%   N13:20  LP_BLEND_GAS_WRN_SP  "CONFIG Blend Gas Low Press Warning Setpoint" %
%   N13:0  REGEN_STATE  "<datalog> STATE The current state of the regen process" %
%   N9:34  REGEN_H2_REDUCTION  "STATE Regen Running" %
%   N13:1  REGEN_BUFFER  "STATE The buffered, previous state of the regen process" %
%   N7:4/11  LP_BLEND_GAS_WRN_EN  "CONFIG Blend Gas Low Press Warning Enable" %
%   T4:60  LP_BLEND_GAS_WRN_TMR %
% Rung: 7 %
SOR XIC T4:60/DN OTE N13:16/4 EOR
%   T4:60  LP_BLEND_GAS_WRN_TMR %
%   N13:16/4  LP_BLEND_GAS_WARN %
% Rung: 8 %
% High Pressure Blend Gas Alarm %
SOR GEQ N20:1 N13:21 NEQ I:5.2 21000 BST EQU N13:0 N9:34 NXB EQU N13:1 N9:34 BND XIC N7:2/12 XIO N13:14/3 XIO N13:16/3 TON T4:61 1.0 10 0 EOR
%   N20:1  MIX_PANEL_PSIG  "<datalog>" %
%   N13:21  HP_BLEND_GAS_ALM_SP  "CONFIG Blend Gas High Press Alarm Setpoint" %
%   I:5.2  MIX_PANEL_PX_READING  "PX-3" %
%   N13:0  REGEN_STATE  "<datalog> STATE The current state of the regen process" %
%   N9:34  REGEN_H2_REDUCTION  "STATE Regen Running" %
%   N13:1  REGEN_BUFFER  "STATE The buffered, previous state of the regen process" %
%   N7:2/12  HP_BLEND_GAS_ALM_EN  "CONFIG Blend Gas High Press Alarm Enable" %
%   N13:14/3  OPEN_PX3_ALARM %
%   N13:16/3  OPEN_PX3_WARN %
%   T4:61  HP_BLEND_GAS_ALM_TMR %
% Rung: 9 %
SOR BST XIC T4:61/DN NXB XIC N13:14/5 XIO B31:4/0 BND OTE N13:14/5 EOR
%   T4:61  HP_BLEND_GAS_ALM_TMR %
%   N13:14/5  HP_BLEND_GAS_ALARM %
%   B31:4/0  REGEN_RESUME  "COMMAND HMI Regen Resume" %

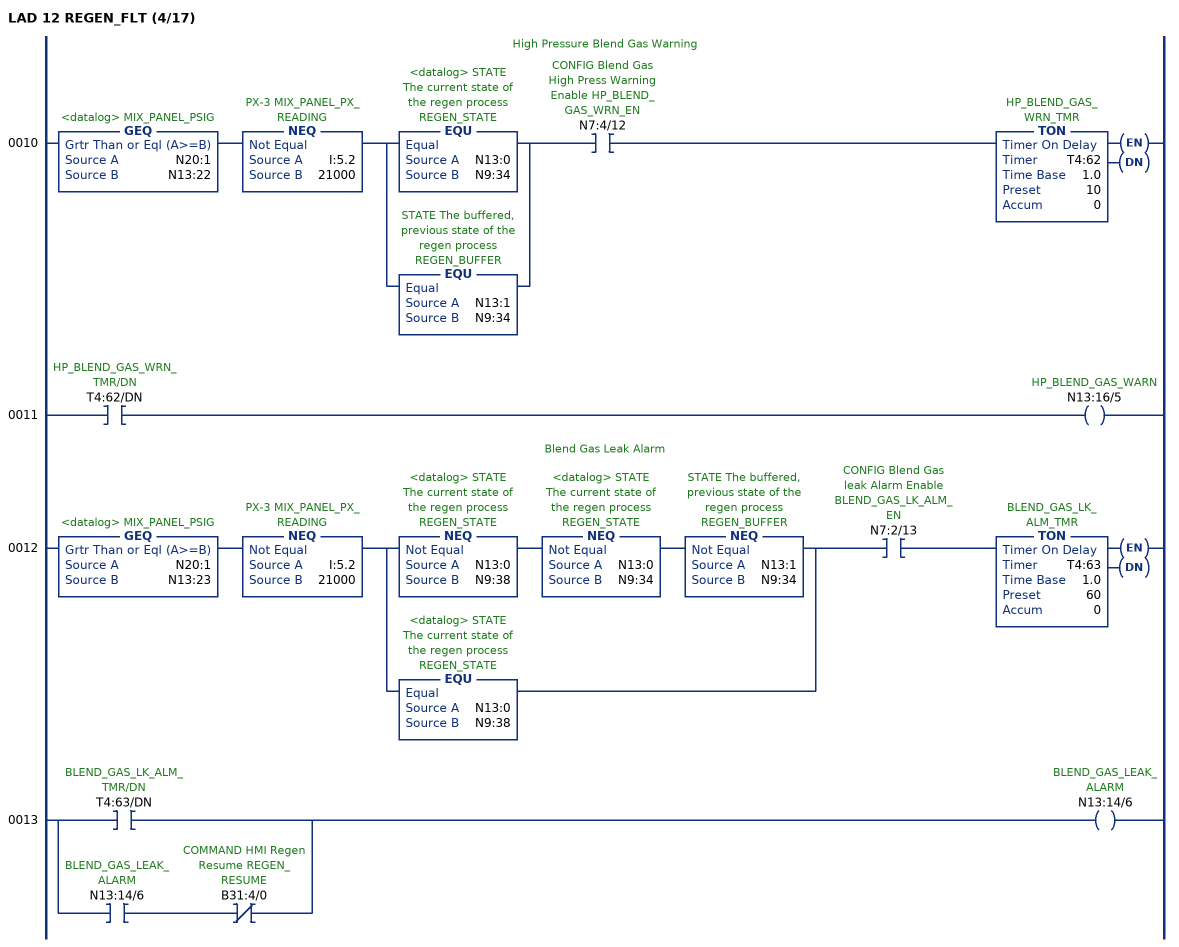
% Rung: 10 %
% High Pressure Blend Gas Warning %
SOR GEQ N20:1 N13:22 NEQ I:5.2 21000 BST EQU N13:0 N9:34 NXB EQU N13:1 N9:34 BND XIC N7:4/12 TON T4:62 1.0 10 0 EOR
%   N20:1  MIX_PANEL_PSIG  "<datalog>" %
%   N13:22  HP_BLEND_GAS_WRN_SP  "CONFIG Blend Gas High Press Warning Setpoint" %
%   I:5.2  MIX_PANEL_PX_READING  "PX-3" %
%   N13:0  REGEN_STATE  "<datalog> STATE The current state of the regen process" %
%   N9:34  REGEN_H2_REDUCTION  "STATE Regen Running" %
%   N13:1  REGEN_BUFFER  "STATE The buffered, previous state of the regen process" %
%   N7:4/12  HP_BLEND_GAS_WRN_EN  "CONFIG Blend Gas High Press Warning Enable" %
%   T4:62  HP_BLEND_GAS_WRN_TMR %
% Rung: 11 %
SOR XIC T4:62/DN OTE N13:16/5 EOR
%   T4:62  HP_BLEND_GAS_WRN_TMR %
%   N13:16/5  HP_BLEND_GAS_WARN %
% Rung: 12 %
% Blend Gas Leak Alarm %
SOR GEQ N20:1 N13:23 NEQ I:5.2 21000 BST NEQ N13:0 N9:38 NEQ N13:0 N9:34 NEQ N13:1 N9:34 NXB EQU N13:0 N9:38 BND XIC N7:2/13 TON T4:63 1.0 60 0 EOR
%   N20:1  MIX_PANEL_PSIG  "<datalog>" %
%   N13:23  BLEND_GAS_LK_ALM_SP  "CONFIG Blend Gas Leak Alarm Setpoint" %
%   I:5.2  MIX_PANEL_PX_READING  "PX-3" %
%   N13:0  REGEN_STATE  "<datalog> STATE The current state of the regen process" %
%   N9:38  REGEN_PURGE  "STATE Regen Hot Purge" %
%   N9:34  REGEN_H2_REDUCTION  "STATE Regen Running" %
%   N13:1  REGEN_BUFFER  "STATE The buffered, previous state of the regen process" %
%   N7:2/13  BLEND_GAS_LK_ALM_EN  "CONFIG Blend Gas leak Alarm Enable" %
%   T4:63  BLEND_GAS_LK_ALM_TMR %
% Rung: 13 %
SOR BST XIC T4:63/DN NXB XIC N13:14/6 XIO B31:4/0 BND OTE N13:14/6 EOR
%   T4:63  BLEND_GAS_LK_ALM_TMR %
%   N13:14/6  BLEND_GAS_LEAK_ALARM %
%   B31:4/0  REGEN_RESUME  "COMMAND HMI Regen Resume" %

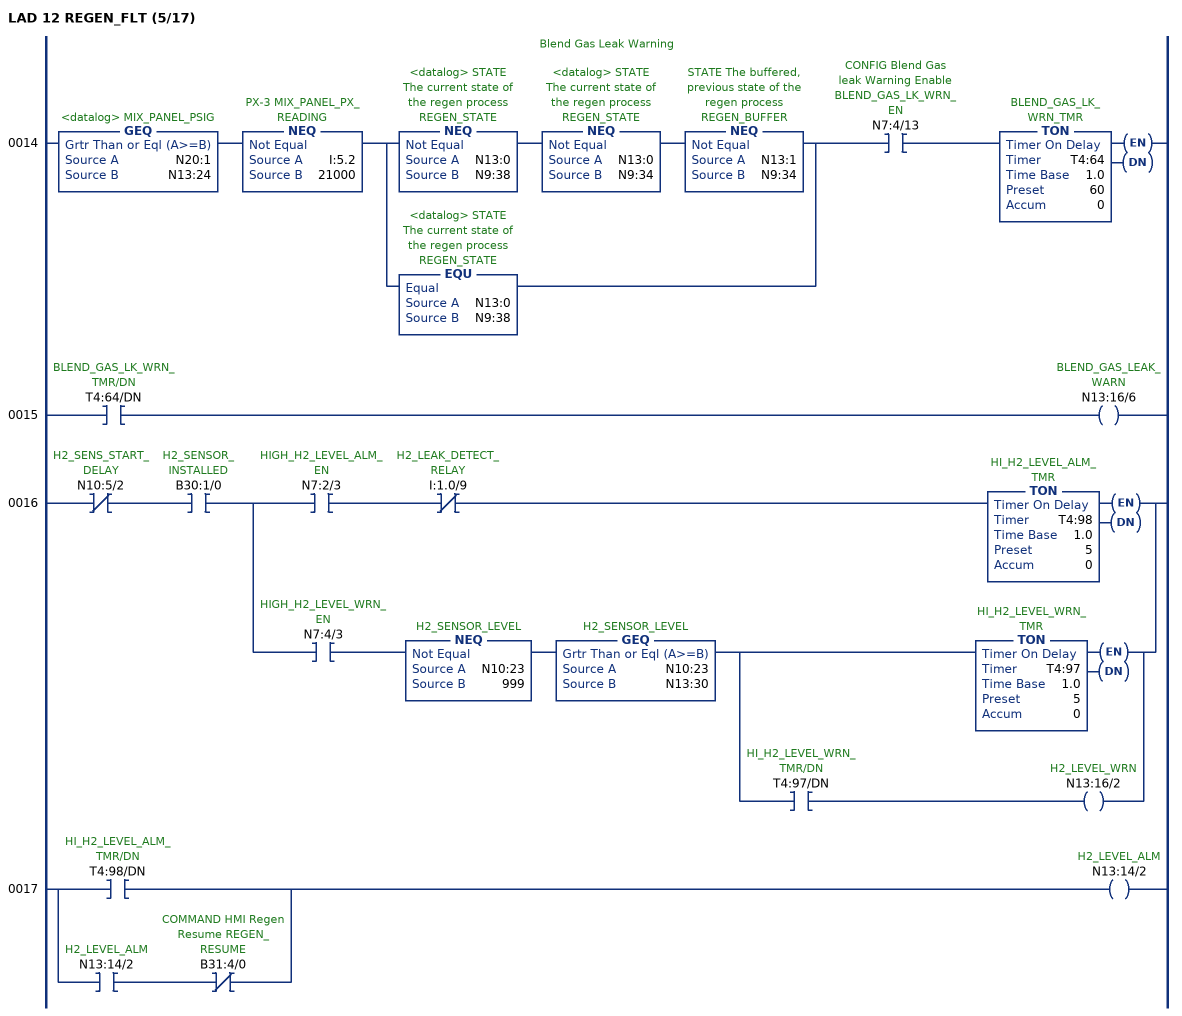
% Rung: 14 %
% Blend Gas Leak Warning %
SOR GEQ N20:1 N13:24 NEQ I:5.2 21000 BST NEQ N13:0 N9:38 NEQ N13:0 N9:34 NEQ N13:1 N9:34 NXB EQU N13:0 N9:38 BND XIC N7:4/13 TON T4:64 1.0 60 0 EOR
%   N20:1  MIX_PANEL_PSIG  "<datalog>" %
%   N13:24  BLEND_GAS_LK_WRN_SP  "CONFIG Blend Gas Leak Warning Setpoint" %
%   I:5.2  MIX_PANEL_PX_READING  "PX-3" %
%   N13:0  REGEN_STATE  "<datalog> STATE The current state of the regen process" %
%   N9:38  REGEN_PURGE  "STATE Regen Hot Purge" %
%   N9:34  REGEN_H2_REDUCTION  "STATE Regen Running" %
%   N13:1  REGEN_BUFFER  "STATE The buffered, previous state of the regen process" %
%   N7:4/13  BLEND_GAS_LK_WRN_EN  "CONFIG Blend Gas leak Warning Enable" %
%   T4:64  BLEND_GAS_LK_WRN_TMR %
% Rung: 15 %
SOR XIC T4:64/DN OTE N13:16/6 EOR
%   T4:64  BLEND_GAS_LK_WRN_TMR %
%   N13:16/6  BLEND_GAS_LEAK_WARN %
% Rung: 16 %
SOR XIO N10:5/2 XIC B30:1/0 BST XIC N7:2/3 XIO I:1.0/9 TON T4:98 1.0 5 0 NXB XIC N7:4/3 NEQ N10:23 999 GEQ N10:23 N13:30 BST TON T4:97 1.0 5 0 NXB XIC T4:97/DN OTE N13:16/2 BND BND EOR
%   N10:5/2  H2_SENS_START_DELAY %
%   B30:1/0  H2_SENSOR_INSTALLED %
%   N7:2/3  HIGH_H2_LEVEL_ALM_EN %
%   I:1.0/9  H2_LEAK_DETECT_RELAY %
%   T4:98  HI_H2_LEVEL_ALM_TMR %
%   N7:4/3  HIGH_H2_LEVEL_WRN_EN %
%   N10:23  H2_SENSOR_LEVEL %
%   N13:30  HIGH_H2_LEVEL_WRN_SP %
%   T4:97  HI_H2_LEVEL_WRN_TMR %
%   N13:16/2  H2_LEVEL_WRN %
% Rung: 17 %
SOR BST XIC T4:98/DN NXB XIC N13:14/2 XIO B31:4/0 BND OTE N13:14/2 EOR
%   T4:98  HI_H2_LEVEL_ALM_TMR %
%   N13:14/2  H2_LEVEL_ALM %
%   B31:4/0  REGEN_RESUME  "COMMAND HMI Regen Resume" %

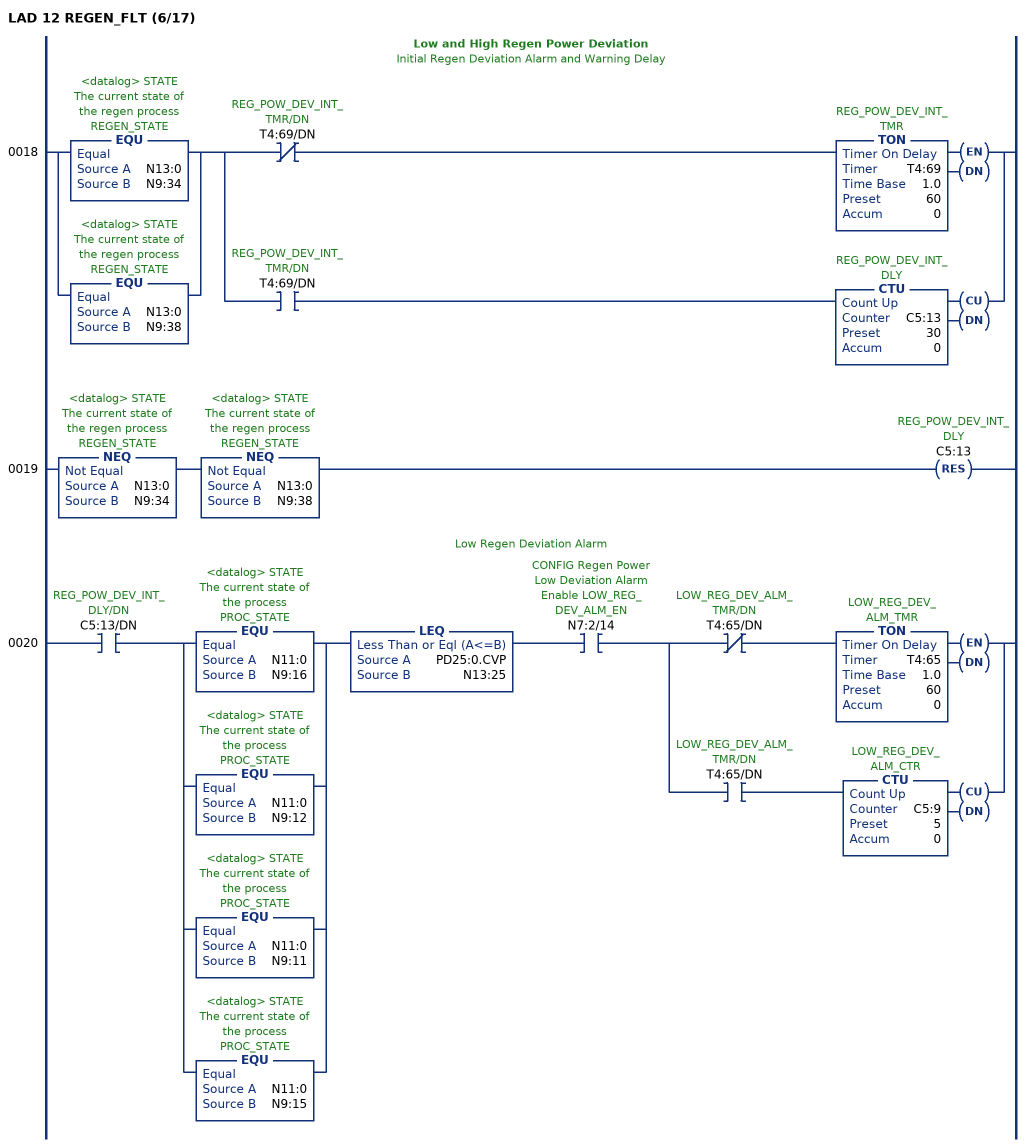
% Rung: 18 %
% TITLE: Low and High Regen Power Deviation %
% Initial Regen Deviation Alarm and Warning Delay %
SOR BST EQU N13:0 N9:34 NXB EQU N13:0 N9:38 BND BST XIO T4:69/DN TON T4:69 1.0 60 0 NXB XIC T4:69/DN CTU C5:13 30 0 BND EOR
%   N13:0  REGEN_STATE  "<datalog> STATE The current state of the regen process" %
%   N9:34  REGEN_H2_REDUCTION  "STATE Regen Running" %
%   N9:38  REGEN_PURGE  "STATE Regen Hot Purge" %
%   T4:69  REG_POW_DEV_INT_TMR %
%   C5:13  REG_POW_DEV_INT_DLY %
% Rung: 19 %
SOR NEQ N13:0 N9:34 NEQ N13:0 N9:38 RES C5:13 EOR
%   N13:0  REGEN_STATE  "<datalog> STATE The current state of the regen process" %
%   N9:34  REGEN_H2_REDUCTION  "STATE Regen Running" %
%   N9:38  REGEN_PURGE  "STATE Regen Hot Purge" %
%   C5:13  REG_POW_DEV_INT_DLY %
% Rung: 20 %
% Low Regen Deviation Alarm %
SOR XIC C5:13/DN BST EQU N11:0 N9:16 NXB EQU N11:0 N9:12 NXB EQU N11:0 N9:11 NXB EQU N11:0 N9:15 BND LEQ PD25:0.CVP N13:25 XIC N7:2/14 BST XIO T4:65/DN TON T4:65 1.0 60 0 NXB XIC T4:65/DN CTU C5:9 5 0 BND EOR
%   C5:13  REG_POW_DEV_INT_DLY %
%   N11:0  PROC_STATE  "<datalog> STATE The current state of the process" %
%   N9:16  PROC_REGEN_D  "STATE Process Regen D" %
%   N9:12  PROC_REGEN_A  "STATE Process Regen A" %
%   N9:11  PROC_REGEN_B  "STATE Process Regen B" %
%   N9:15  PROC_REGEN_C  "STATE Process Regen C" %
%   N13:25  LOW_REG_DEV_ALM_SP  "CONFIG Regen Power Low Deviation Alarm Setpoint" %
%   N7:2/14  LOW_REG_DEV_ALM_EN  "CONFIG Regen Power Low Deviation Alarm Enable" %
%   T4:65  LOW_REG_DEV_ALM_TMR %
%   C5:9  LOW_REG_DEV_ALM_CTR %

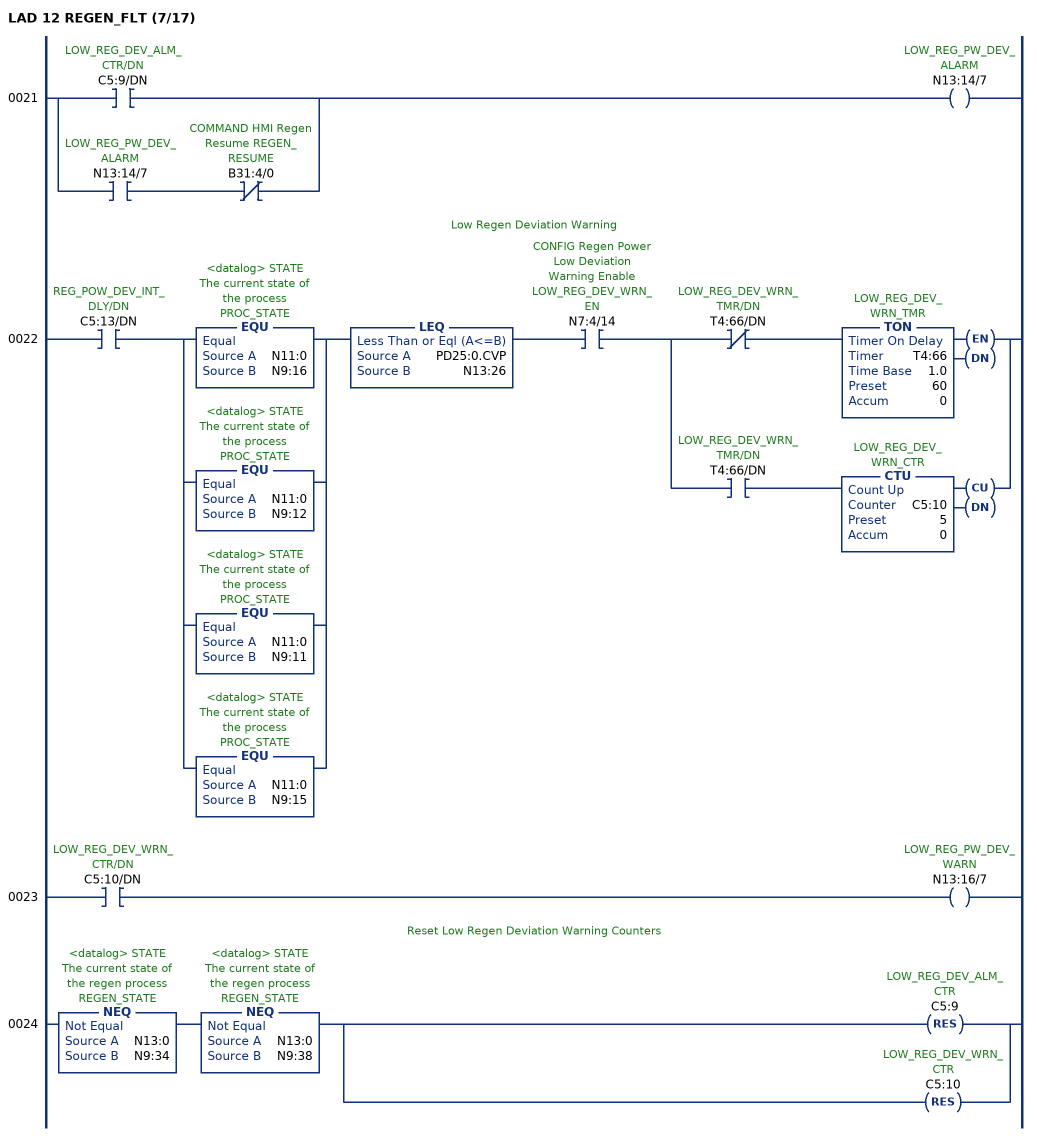
% Rung: 21 %
SOR BST XIC C5:9/DN NXB XIC N13:14/7 XIO B31:4/0 BND OTE N13:14/7 EOR
%   C5:9  LOW_REG_DEV_ALM_CTR %
%   N13:14/7  LOW_REG_PW_DEV_ALARM %
%   B31:4/0  REGEN_RESUME  "COMMAND HMI Regen Resume" %
% Rung: 22 %
% Low Regen Deviation Warning %
SOR XIC C5:13/DN BST EQU N11:0 N9:16 NXB EQU N11:0 N9:12 NXB EQU N11:0 N9:11 NXB EQU N11:0 N9:15 BND LEQ PD25:0.CVP N13:26 XIC N7:4/14 BST XIO T4:66/DN TON T4:66 1.0 60 0 NXB XIC T4:66/DN CTU C5:10 5 0 BND EOR
%   C5:13  REG_POW_DEV_INT_DLY %
%   N11:0  PROC_STATE  "<datalog> STATE The current state of the process" %
%   N9:16  PROC_REGEN_D  "STATE Process Regen D" %
%   N9:12  PROC_REGEN_A  "STATE Process Regen A" %
%   N9:11  PROC_REGEN_B  "STATE Process Regen B" %
%   N9:15  PROC_REGEN_C  "STATE Process Regen C" %
%   N13:26  LOW_REG_DEV_WRN_SP  "CONFIG Regen Power Low Deviation Warning Setpoint" %
%   N7:4/14  LOW_REG_DEV_WRN_EN  "CONFIG Regen Power Low Deviation Warning Enable" %
%   T4:66  LOW_REG_DEV_WRN_TMR %
%   C5:10  LOW_REG_DEV_WRN_CTR %
% Rung: 23 %
SOR XIC C5:10/DN OTE N13:16/7 EOR
%   C5:10  LOW_REG_DEV_WRN_CTR %
%   N13:16/7  LOW_REG_PW_DEV_WARN %
% Rung: 24 %
% Reset Low Regen Deviation Warning Counters %
SOR NEQ N13:0 N9:34 NEQ N13:0 N9:38 BST RES C5:9 NXB RES C5:10 BND EOR
%   N13:0  REGEN_STATE  "<datalog> STATE The current state of the regen process" %
%   N9:34  REGEN_H2_REDUCTION  "STATE Regen Running" %
%   N9:38  REGEN_PURGE  "STATE Regen Hot Purge" %
%   C5:9  LOW_REG_DEV_ALM_CTR %
%   C5:10  LOW_REG_DEV_WRN_CTR %

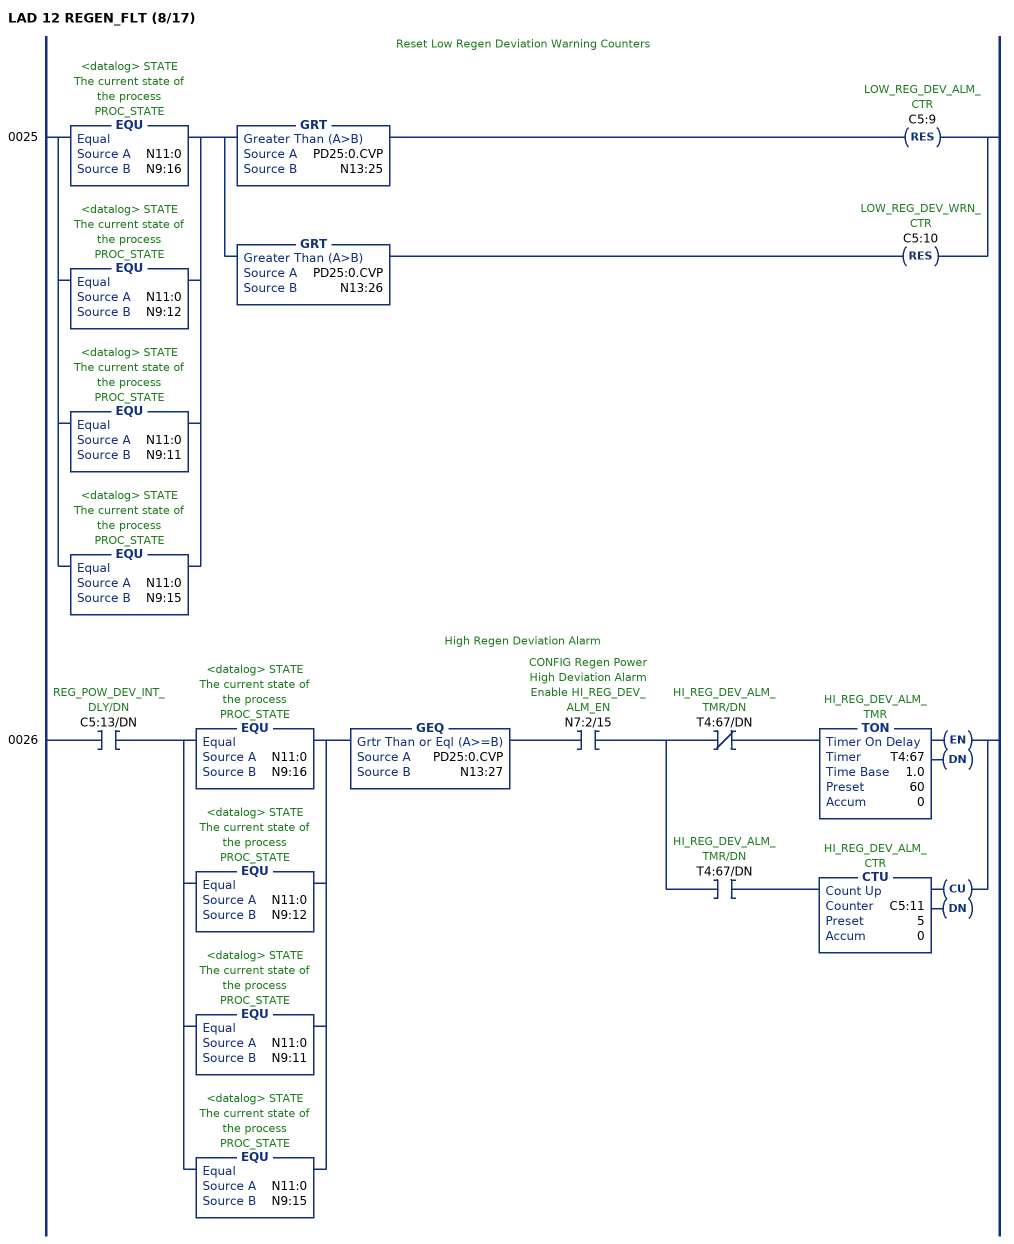
% Rung: 25 %
% Reset Low Regen Deviation Warning Counters %
SOR BST EQU N11:0 N9:16 NXB EQU N11:0 N9:12 NXB EQU N11:0 N9:11 NXB EQU N11:0 N9:15 BND BST GRT PD25:0.CVP N13:25 RES C5:9 NXB GRT PD25:0.CVP N13:26 RES C5:10 BND EOR
%   N11:0  PROC_STATE  "<datalog> STATE The current state of the process" %
%   N9:16  PROC_REGEN_D  "STATE Process Regen D" %
%   N9:12  PROC_REGEN_A  "STATE Process Regen A" %
%   N9:11  PROC_REGEN_B  "STATE Process Regen B" %
%   N9:15  PROC_REGEN_C  "STATE Process Regen C" %
%   N13:25  LOW_REG_DEV_ALM_SP  "CONFIG Regen Power Low Deviation Alarm Setpoint" %
%   C5:9  LOW_REG_DEV_ALM_CTR %
%   N13:26  LOW_REG_DEV_WRN_SP  "CONFIG Regen Power Low Deviation Warning Setpoint" %
%   C5:10  LOW_REG_DEV_WRN_CTR %
% Rung: 26 %
% High Regen Deviation Alarm %
SOR XIC C5:13/DN BST EQU N11:0 N9:16 NXB EQU N11:0 N9:12 NXB EQU N11:0 N9:11 NXB EQU N11:0 N9:15 BND GEQ PD25:0.CVP N13:27 XIC N7:2/15 BST XIO T4:67/DN TON T4:67 1.0 60 0 NXB XIC T4:67/DN CTU C5:11 5 0 BND EOR
%   C5:13  REG_POW_DEV_INT_DLY %
%   N11:0  PROC_STATE  "<datalog> STATE The current state of the process" %
%   N9:16  PROC_REGEN_D  "STATE Process Regen D" %
%   N9:12  PROC_REGEN_A  "STATE Process Regen A" %
%   N9:11  PROC_REGEN_B  "STATE Process Regen B" %
%   N9:15  PROC_REGEN_C  "STATE Process Regen C" %
%   N13:27  HI_REG_DEV_ALM_SP  "CONFIG Regen Power High Deviation Alarm Setpoint" %
%   N7:2/15  HI_REG_DEV_ALM_EN  "CONFIG Regen Power High Deviation Alarm Enable" %
%   T4:67  HI_REG_DEV_ALM_TMR %
%   C5:11  HI_REG_DEV_ALM_CTR %

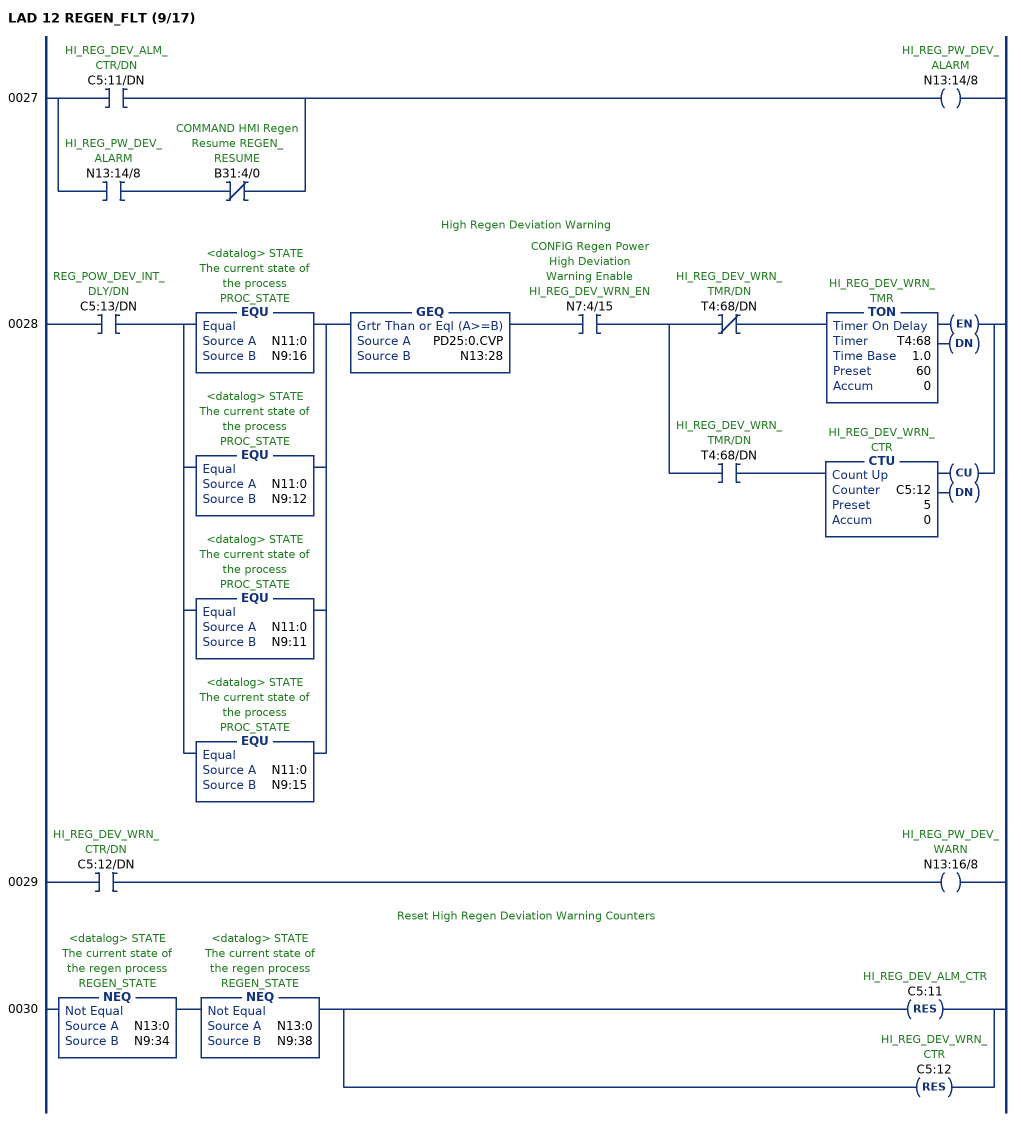
% Rung: 27 %
SOR BST XIC C5:11/DN NXB XIC N13:14/8 XIO B31:4/0 BND OTE N13:14/8 EOR
%   C5:11  HI_REG_DEV_ALM_CTR %
%   N13:14/8  HI_REG_PW_DEV_ALARM %
%   B31:4/0  REGEN_RESUME  "COMMAND HMI Regen Resume" %
% Rung: 28 %
% High Regen Deviation Warning %
SOR XIC C5:13/DN BST EQU N11:0 N9:16 NXB EQU N11:0 N9:12 NXB EQU N11:0 N9:11 NXB EQU N11:0 N9:15 BND GEQ PD25:0.CVP N13:28 XIC N7:4/15 BST XIO T4:68/DN TON T4:68 1.0 60 0 NXB XIC T4:68/DN CTU C5:12 5 0 BND EOR
%   C5:13  REG_POW_DEV_INT_DLY %
%   N11:0  PROC_STATE  "<datalog> STATE The current state of the process" %
%   N9:16  PROC_REGEN_D  "STATE Process Regen D" %
%   N9:12  PROC_REGEN_A  "STATE Process Regen A" %
%   N9:11  PROC_REGEN_B  "STATE Process Regen B" %
%   N9:15  PROC_REGEN_C  "STATE Process Regen C" %
%   N13:28  HI_REG_DEV_WRN_SP  "CONFIG Regen Power High Deviation Warning Setpoint" %
%   N7:4/15  HI_REG_DEV_WRN_EN  "CONFIG Regen Power High Deviation Warning Enable" %
%   T4:68  HI_REG_DEV_WRN_TMR %
%   C5:12  HI_REG_DEV_WRN_CTR %
% Rung: 29 %
SOR XIC C5:12/DN OTE N13:16/8 EOR
%   C5:12  HI_REG_DEV_WRN_CTR %
%   N13:16/8  HI_REG_PW_DEV_WARN %
% Rung: 30 %
% Reset High Regen Deviation Warning Counters %
SOR NEQ N13:0 N9:34 NEQ N13:0 N9:38 BST RES C5:11 NXB RES C5:12 BND EOR
%   N13:0  REGEN_STATE  "<datalog> STATE The current state of the regen process" %
%   N9:34  REGEN_H2_REDUCTION  "STATE Regen Running" %
%   N9:38  REGEN_PURGE  "STATE Regen Hot Purge" %
%   C5:11  HI_REG_DEV_ALM_CTR %
%   C5:12  HI_REG_DEV_WRN_CTR %

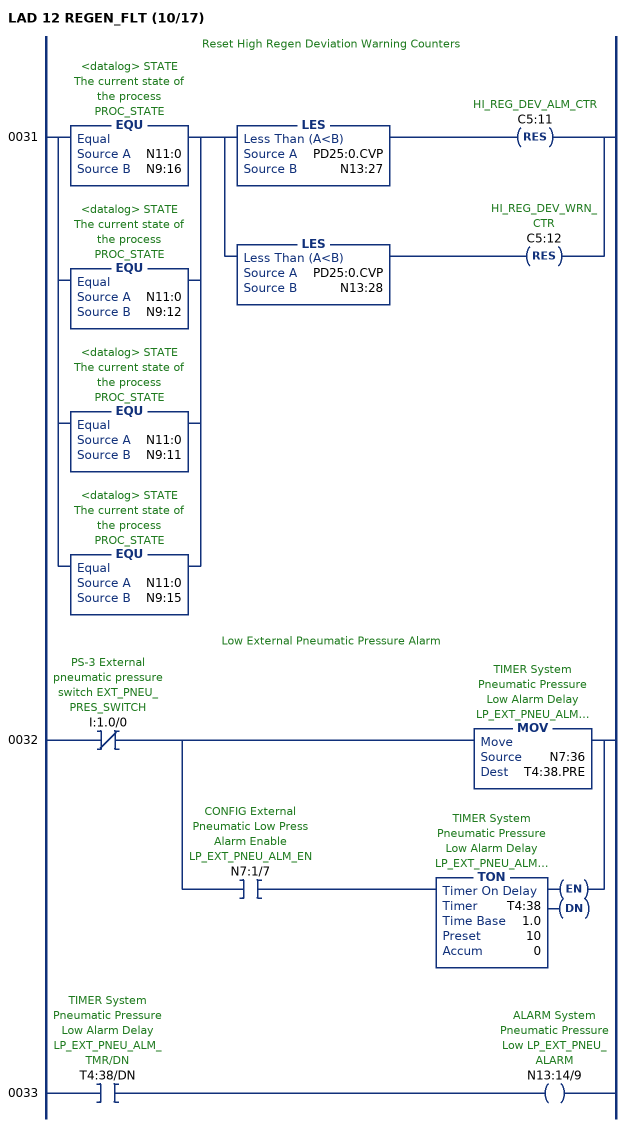
% Rung: 31 %
% Reset High Regen Deviation Warning Counters %
SOR BST EQU N11:0 N9:16 NXB EQU N11:0 N9:12 NXB EQU N11:0 N9:11 NXB EQU N11:0 N9:15 BND BST LES PD25:0.CVP N13:27 RES C5:11 NXB LES PD25:0.CVP N13:28 RES C5:12 BND EOR
%   N11:0  PROC_STATE  "<datalog> STATE The current state of the process" %
%   N9:16  PROC_REGEN_D  "STATE Process Regen D" %
%   N9:12  PROC_REGEN_A  "STATE Process Regen A" %
%   N9:11  PROC_REGEN_B  "STATE Process Regen B" %
%   N9:15  PROC_REGEN_C  "STATE Process Regen C" %
%   N13:27  HI_REG_DEV_ALM_SP  "CONFIG Regen Power High Deviation Alarm Setpoint" %
%   C5:11  HI_REG_DEV_ALM_CTR %
%   N13:28  HI_REG_DEV_WRN_SP  "CONFIG Regen Power High Deviation Warning Setpoint" %
%   C5:12  HI_REG_DEV_WRN_CTR %
% Rung: 32 %
% Low External Pneumatic Pressure Alarm %
SOR XIO I:1.0/0 BST MOV N7:36 T4:38.PRE NXB XIC N7:1/7 TON T4:38 1.0 10 0 BND EOR
%   I:1.0/0  EXT_PNEU_PRES_SWITCH  "PS-3 External pneumatic pressure switch" %
%   N7:36  LP_EXT_PNEU_ALM_DLY  "CONFIG External Pneumatic Low Press Alarm Delay" %
%   T4:38  LP_EXT_PNEU_ALM_TMR  "TIMER System Pneumatic Pressure Low Alarm Delay" %
%   N7:1/7  LP_EXT_PNEU_ALM_EN  "CONFIG External Pneumatic Low Press Alarm Enable" %
% Rung: 33 %
SOR XIC T4:38/DN OTE N13:14/9 EOR
%   T4:38  LP_EXT_PNEU_ALM_TMR  "TIMER System Pneumatic Pressure Low Alarm Delay" %
%   N13:14/9  LP_EXT_PNEU_ALARM  "ALARM System Pneumatic Pressure Low" %

